LIN {X 80.299,Y 11.763,Z 59.815,A 180.000,B 0.000,C 180.000} C_DIS
LIN {X 80.187,Y 11.652,Z 59.809,A 180.000,B 0.000,C 180.000} C_DIS
LIN {X 80.132,Y 11.596,Z 59.806,A 180.000,B 0.000,C 180.000} C_DIS
LIN {X 80.020,Y 11.485,Z 59.801,A 180.000,B 0.000,C 180.000} C_DIS
LIN {X 79.853,Y 11.318,Z 59.793,A 180.000,B 0.000,C 180.000} C_DIS
LIN {X 79.742,Y 11.206,Z 59.787,A 180.000,B 0.000,C 180.000} C_DIS
LIN {X 79.686,Y 11.151,Z 59.785,A 180.000,B 0.000,C 180.000} C_DIS
LIN {X 79.575,Y 11.039,Z 59.779,A 180.000,B 0.000,C 180.000} C_DIS
LIN {X 79.408,Y 10.872,Z 59.771,A 180.000,B 0.000,C 180.000} C_DIS
LIN {X 79.296,Y 10.761,Z 59.765,A 180.000,B 0.000,C 180.000} C_DIS
LIN {X 79.241,Y 10.705,Z 59.763,A 180.000,B 0.000,C 180.000} C_DIS
LIN {X 79.183,Y 10.652,Z 59.760,A 180.000,B 0.000,C 180.000} C_DIS
LIN {X 79.124,Y 10.599,Z 59.757,A 180.000,B 0.000,C 180.000} C_DIS
LIN {X 79.063,Y 10.549,Z 59.754,A 180.000,B 0.000,C 180.000} C_DIS
LIN {X 79.001,Y 10.501,Z 59.752,A 180.000,B 0.000,C 180.000} C_DIS
LIN {X 78.938,Y 10.455,Z 59.749,A 180.000,B 0.000,C 180.000} C_DIS
LIN {X 78.872,Y 10.410,Z 59.746,A 180.000,B 0.000,C 180.000} C_DIS
LIN {X 78.806,Y 10.368,Z 59.743,A 180.000,B 0.000,C 180.000} C_DIS
LIN {X 78.738,Y 10.328,Z 59.741,A 180.000,B 0.000,C 180.000} C_DIS
LIN {X 78.669,Y 10.290,Z 59.738,A 180.000,B 0.000,C 180.000} C_DIS
LIN {X 78.599,Y 10.254,Z 59.735,A 180.000,B 0.000,C 180.000} C_DIS
LIN {X 78.528,Y 10.221,Z 59.732,A 180.000,B 0.000,C 180.000} C_DIS
LIN {X 78.455,Y 10.190,Z 59.730,A 180.000,B 0.000,C 180.000} C_DIS
LIN {X 78.382,Y 10.161,Z 59.727,A 180.000,B 0.000,C 180.000} C_DIS
LIN {X 78.308,Y 10.134,Z 59.724,A 180.000,B 0.000,C 180.000} C_DIS
LIN {X 78.233,Y 10.110,Z 59.721,A 180.000,B 0.000,C 180.000} C_DIS
LIN {X 78.157,Y 10.088,Z 59.719,A 180.000,B 0.000,C 180.000} C_DIS
LIN {X 78.081,Y 10.068,Z 59.716,A 180.000,B 0.000,C 180.000} C_DIS
LIN {X 78.004,Y 10.051,Z 59.713,A 180.000,B 0.000,C 180.000} C_DIS
LIN {X 77.927,Y 10.037,Z 59.710,A 180.000,B 0.000,C 180.000} C_DIS
LIN {X 77.849,Y 10.024,Z 59.708,A 180.000,B 0.000,C 180.000} C_DIS
LIN {X 77.771,Y 10.015,Z 59.705,A 180.000,B 0.000,C 180.000} C_DIS
LIN {X 77.692,Y 10.007,Z 59.702,A 180.000,B 0.000,C 180.000} C_DIS
LIN {X 77.614,Y 10.003,Z 59.699,A 180.000,B 0.000,C 180.000} C_DIS
LIN {X 77.535,Y 10.000,Z 59.697,A 180.000,B 0.000,C 180.000} C_DIS
LIN {X 77.456,Y 10.000,Z 59.694,A 180.000,B 0.000,C 180.000} C_DIS
LIN {X 77.377,Y 10.003,Z 59.691,A 180.000,B 0.000,C 180.000} C_DIS
LIN {X 77.299,Y 10.008,Z 59.688,A 180.000,B 0.000,C 180.000} C_DIS
LIN {X 77.220,Y 10.016,Z 59.686,A 180.000,B 0.000,C 180.000} C_DIS
LIN {X 77.142,Y 10.026,Z 59.683,A 180.000,B 0.000,C 180.000} C_DIS
LIN {X 77.065,Y 10.038,Z 59.680,A 180.000,B 0.000,C 180.000} C_DIS
LIN {X 76.987,Y 10.053,Z 59.677,A 180.000,B 0.000,C 180.000} C_DIS
LIN {X 76.910,Y 10.071,Z 59.675,A 180.000,B 0.000,C 180.000} C_DIS
LIN {X 76.834,Y 10.090,Z 59.672,A 180.000,B 0.000,C 180.000} C_DIS
LIN {X 76.759,Y 10.112,Z 59.669,A 180.000,B 0.000,C 180.000} C_DIS
LIN {X 76.684,Y 10.137,Z 59.666,A 180.000,B 0.000,C 180.000} C_DIS
LIN {X 76.610,Y 10.164,Z 59.664,A 180.000,B 0.000,C 180.000} C_DIS
LIN {X 76.537,Y 10.193,Z 59.661,A 180.000,B 0.000,C 180.000} C_DIS
LIN {X 76.464,Y 10.225,Z 59.658,A 180.000,B 0.000,C 180.000} C_DIS
LIN {X 76.393,Y 10.258,Z 59.655,A 180.000,B 0.000,C 180.000} C_DIS
LIN {X 76.323,Y 10.294,Z 59.653,A 180.000,B 0.000,C 180.000} C_DIS
LIN {X 76.254,Y 10.332,Z 59.650,A 180.000,B 0.000,C 180.000} C_DIS
LIN {X 76.187,Y 10.373,Z 59.647,A 180.000,B 0.000,C 180.000} C_DIS
LIN {X 76.120,Y 10.415,Z 59.644,A 180.000,B 0.000,C 180.000} C_DIS
LIN {X 76.055,Y 10.460,Z 59.642,A 180.000,B 0.000,C 180.000} C_DIS
LIN {X 75.992,Y 10.506,Z 59.639,A 180.000,B 0.000,C 180.000} C_DIS
LIN {X 75.930,Y 10.555,Z 59.636,A 180.000,B 0.000,C 180.000} C_DIS
LIN {X 75.869,Y 10.605,Z 59.633,A 180.000,B 0.000,C 180.000} C_DIS
LIN {X 75.810,Y 10.658,Z 59.631,A 180.000,B 0.000,C 180.000} C_DIS
LIN {X 75.753,Y 10.712,Z 59.628,A 180.000,B 0.000,C 180.000} C_DIS
LIN {X 75.697,Y 10.767,Z 59.625,A 180.000,B 0.000,C 180.000} C_DIS
LIN {X 75.140,Y 11.324,Z 59.598,A 180.000,B 0.000,C 180.000} C_DIS
LIN {X 74.973,Y 11.491,Z 59.589,A 180.000,B 0.000,C 180.000} C_DIS
LIN {X 74.751,Y 11.714,Z 59.578,A 180.000,B 0.000,C 180.000} C_DIS
LIN {X 74.472,Y 11.992,Z 59.565,A 180.000,B 0.000,C 180.000} C_DIS
LIN {X 74.138,Y 12.326,Z 59.548,A 180.000,B 0.000,C 180.000} C_DIS
LIN {X 72.857,Y 13.607,Z 59.485,A 180.000,B 0.000,C 180.000} C_DIS
LIN {X 70.741,Y 15.723,Z 59.380,A 180.000,B 0.000,C 180.000} C_DIS
LIN {X 70.630,Y 15.834,Z 59.375,A 180.000,B 0.000,C 180.000} C_DIS
LIN {X 70.296,Y 16.169,Z 59.358,A 180.000,B 0.000,C 180.000} C_DIS
LIN {X 70.185,Y 16.280,Z 59.353,A 180.000,B 0.000,C 180.000} C_DIS
LIN {X 69.850,Y 16.614,Z 59.336,A 180.000,B 0.000,C 180.000} C_DIS
LIN {X 69.795,Y 16.670,Z 59.334,A 180.000,B 0.000,C 180.000} C_DIS
LIN {X 69.683,Y 16.781,Z 59.328,A 180.000,B 0.000,C 180.000} C_DIS
LIN {X 69.349,Y 17.115,Z 59.312,A 180.000,B 0.000,C 180.000} C_DIS
LIN {X 69.238,Y 17.227,Z 59.306,A 180.000,B 0.000,C 180.000} C_DIS
LIN {X 68.904,Y 17.561,Z 59.290,A 180.000,B 0.000,C 180.000} C_DIS
LIN {X 68.792,Y 17.672,Z 59.284,A 180.000,B 0.000,C 180.000} C_DIS
LIN {X 68.625,Y 17.839,Z 59.276,A 180.000,B 0.000,C 180.000} C_DIS
LIN {X 68.514,Y 17.951,Z 59.270,A 180.000,B 0.000,C 180.000} C_DIS
LIN {X 68.458,Y 18.006,Z 59.268,A 180.000,B 0.000,C 180.000} C_DIS
LIN {X 68.347,Y 18.118,Z 59.262,A 180.000,B 0.000,C 180.000} C_DIS
LIN {X 68.180,Y 18.285,Z 59.254,A 180.000,B 0.000,C 180.000} C_DIS
LIN {X 68.068,Y 18.396,Z 59.248,A 180.000,B 0.000,C 180.000} C_DIS
LIN {X 68.013,Y 18.452,Z 59.246,A 180.000,B 0.000,C 180.000} C_DIS
LIN {X 67.901,Y 18.563,Z 59.240,A 180.000,B 0.000,C 180.000} C_DIS
LIN {X 67.734,Y 18.730,Z 59.232,A 180.000,B 0.000,C 180.000} C_DIS
LIN {X 67.623,Y 18.841,Z 59.226,A 180.000,B 0.000,C 180.000} C_DIS
LIN {X 67.567,Y 18.897,Z 59.224,A 180.000,B 0.000,C 180.000} C_DIS
LIN {X 67.456,Y 19.009,Z 59.218,A 180.000,B 0.000,C 180.000} C_DIS
LIN {X 67.289,Y 19.176,Z 59.210,A 180.000,B 0.000,C 180.000} C_DIS
LIN {X 67.178,Y 19.287,Z 59.204,A 180.000,B 0.000,C 180.000} C_DIS
LIN {X 67.122,Y 19.343,Z 59.202,A 180.000,B 0.000,C 180.000} C_DIS
LIN {X 67.010,Y 19.454,Z 59.196,A 180.000,B 0.000,C 180.000} C_DIS
LIN {X 66.899,Y 19.565,Z 59.191,A 180.000,B 0.000,C 180.000} C_DIS
LIN {X 66.788,Y 19.677,Z 59.185,A 180.000,B 0.000,C 180.000} C_DIS
LIN {X 66.676,Y 19.788,Z 59.180,A 180.000,B 0.000,C 180.000} C_DIS
LIN {X 66.565,Y 19.899,Z 59.174,A 180.000,B 0.000,C 180.000} C_DIS
LIN {X 66.454,Y 20.011,Z 59.169,A 180.000,B 0.000,C 180.000} C_DIS
LIN {X 66.342,Y 20.122,Z 59.164,A 180.000,B 0.000,C 180.000} C_DIS
LIN {X 66.287,Y 20.178,Z 59.161,A 180.000,B 0.000,C 180.000} C_DIS
LIN {X 66.231,Y 20.234,Z 59.159,A 180.000,B 0.000,C 180.000} C_DIS
LIN {X 66.175,Y 20.289,Z 59.156,A 180.000,B 0.000,C 180.000} C_DIS
LIN {X 66.120,Y 20.345,Z 59.154,A 180.000,B 0.000,C 180.000} C_DIS
LIN {X 66.064,Y 20.401,Z 59.151,A 180.000,B 0.000,C 180.000} C_DIS
LIN {X 66.008,Y 20.456,Z 59.149,A 180.000,B 0.000,C 180.000} C_DIS
LIN {X 65.897,Y 20.568,Z 59.144,A 180.000,B 0.000,C 180.000} C_DIS
LIN {X 65.785,Y 20.679,Z 59.139,A 180.000,B 0.000,C 180.000} C_DIS
LIN {X 65.674,Y 20.790,Z 59.134,A 180.000,B 0.000,C 180.000} C_DIS
LIN {X 65.563,Y 20.902,Z 59.129,A 180.000,B 0.000,C 180.000} C_DIS
LIN {X 65.451,Y 21.013,Z 59.124,A 180.000,B 0.000,C 180.000} C_DIS
LIN {X 65.340,Y 21.125,Z 59.120,A 180.000,B 0.000,C 180.000} C_DIS
LIN {X 65.229,Y 21.236,Z 59.115,A 180.000,B 0.000,C 180.000} C_DIS
LIN {X 65.117,Y 21.347,Z 59.111,A 180.000,B 0.000,C 180.000} C_DIS
LIN {X 65.006,Y 21.459,Z 59.106,A 180.000,B 0.000,C 180.000} C_DIS
LIN {X 64.894,Y 21.570,Z 59.102,A 180.000,B 0.000,C 180.000} C_DIS
LIN {X 64.783,Y 21.681,Z 59.097,A 180.000,B 0.000,C 180.000} C_DIS
LIN {X 64.672,Y 21.793,Z 59.093,A 180.000,B 0.000,C 180.000} C_DIS
LIN {X 64.560,Y 21.904,Z 59.089,A 180.000,B 0.000,C 180.000} C_DIS
LIN {X 64.449,Y 22.015,Z 59.085,A 180.000,B 0.000,C 180.000} C_DIS
LIN {X 64.338,Y 22.127,Z 59.081,A 180.000,B 0.000,C 180.000} C_DIS
LIN {X 64.226,Y 22.238,Z 59.077,A 180.000,B 0.000,C 180.000} C_DIS
LIN {X 64.115,Y 22.350,Z 59.073,A 180.000,B 0.000,C 180.000} C_DIS
LIN {X 64.004,Y 22.461,Z 59.070,A 180.000,B 0.000,C 180.000} C_DIS
LIN {X 63.892,Y 22.572,Z 59.066,A 180.000,B 0.000,C 180.000} C_DIS
LIN {X 63.781,Y 22.684,Z 59.062,A 180.000,B 0.000,C 180.000} C_DIS
LIN {X 63.669,Y 22.795,Z 59.059,A 180.000,B 0.000,C 180.000} C_DIS
LIN {X 63.558,Y 22.906,Z 59.056,A 180.000,B 0.000,C 180.000} C_DIS
LIN {X 63.447,Y 23.018,Z 59.052,A 180.000,B 0.000,C 180.000} C_DIS
LIN {X 63.335,Y 23.129,Z 59.049,A 180.000,B 0.000,C 180.000} C_DIS
LIN {X 63.224,Y 23.241,Z 59.046,A 180.000,B 0.000,C 180.000} C_DIS
LIN {X 63.113,Y 23.352,Z 59.043,A 180.000,B 0.000,C 180.000} C_DIS
LIN {X 63.001,Y 23.463,Z 59.040,A 180.000,B 0.000,C 180.000} C_DIS
LIN {X 62.890,Y 23.575,Z 59.037,A 180.000,B 0.000,C 180.000} C_DIS
LIN {X 62.778,Y 23.686,Z 59.034,A 180.000,B 0.000,C 180.000} C_DIS
LIN {X 62.667,Y 23.797,Z 59.032,A 180.000,B 0.000,C 180.000} C_DIS
LIN {X 62.556,Y 23.909,Z 59.029,A 180.000,B 0.000,C 180.000} C_DIS
LIN {X 62.444,Y 24.020,Z 59.027,A 180.000,B 0.000,C 180.000} C_DIS
LIN {X 62.222,Y 24.243,Z 59.022,A 180.000,B 0.000,C 180.000} C_DIS
LIN {X 61.999,Y 24.466,Z 59.018,A 180.000,B 0.000,C 180.000} C_DIS
LIN {X 61.776,Y 24.688,Z 59.014,A 180.000,B 0.000,C 180.000} C_DIS
LIN {X 61.553,Y 24.911,Z 59.011,A 180.000,B 0.000,C 180.000} C_DIS
LIN {X 61.331,Y 25.134,Z 59.008,A 180.000,B 0.000,C 180.000} C_DIS
LIN {X 61.108,Y 25.357,Z 59.005,A 180.000,B 0.000,C 180.000} C_DIS
LIN {X 60.885,Y 25.579,Z 59.003,A 180.000,B 0.000,C 180.000} C_DIS
LIN {X 60.662,Y 25.802,Z 59.002,A 180.000,B 0.000,C 180.000} C_DIS
LIN {X 60.440,Y 26.025,Z 59.001,A 180.000,B 0.000,C 180.000} C_DIS
LIN {X 60.217,Y 26.247,Z 59.000,A 180.000,B 0.000,C 180.000} C_DIS
LIN {X 60.053,Y 26.412,Z 59.000,A 180.000,B 0.000,C 180.000} C_DIS
; Cutting Move Starts
LIN {X 10.729,Y 75.735,Z 59.000,A 180.000,B 0.000,C 180.000} C_DIS
LIN {X 10.665,Y 75.802,Z 59.000,A 180.000,B 0.000,C 180.000} C_DIS
LIN {X 10.551,Y 75.935,Z 59.000,A 180.000,B 0.000,C 180.000} C_DIS
LIN {X 10.515,Y 75.980,Z 59.000,A 180.000,B 0.000,C 180.000} C_DIS
LIN {X 10.390,Y 76.159,Z 59.000,A 180.000,B 0.000,C 180.000} C_DIS
LIN {X 10.372,Y 76.188,Z 59.000,A 180.000,B 0.000,C 180.000} C_DIS
LIN {X 10.286,Y 76.338,Z 59.000,A 180.000,B 0.000,C 180.000} C_DIS
LIN {X 10.201,Y 76.517,Z 59.000,A 180.000,B 0.000,C 180.000} C_DIS
LIN {X 10.193,Y 76.537,Z 59.000,A 180.000,B 0.000,C 180.000} C_DIS
LIN {X 10.133,Y 76.696,Z 59.000,A 180.000,B 0.000,C 180.000} C_DIS
LIN {X 10.080,Y 76.874,Z 59.000,A 180.000,B 0.000,C 180.000} C_DIS
LIN {X 10.040,Y 77.053,Z 59.000,A 180.000,B 0.000,C 180.000} C_DIS
LIN {X 10.014,Y 77.232,Z 59.000,A 180.000,B 0.000,C 180.000} C_DIS
LIN {X 10.014,Y 77.233,Z 59.000,A 180.000,B 0.000,C 180.000} C_DIS
LIN {X 10.002,Y 77.411,Z 59.000,A 180.000,B 0.000,C 180.000} C_DIS
LIN {X 10.002,Y 77.589,Z 59.000,A 180.000,B 0.000,C 180.000} C_DIS
LIN {X 10.014,Y 77.767,Z 59.000,A 180.000,B 0.000,C 180.000} C_DIS
LIN {X 10.014,Y 77.768,Z 59.000,A 180.000,B 0.000,C 180.000} C_DIS
LIN {X 10.040,Y 77.947,Z 59.000,A 180.000,B 0.000,C 180.000} C_DIS
LIN {X 10.080,Y 78.126,Z 59.000,A 180.000,B 0.000,C 180.000} C_DIS
LIN {X 10.133,Y 78.304,Z 59.000,A 180.000,B 0.000,C 180.000} C_DIS
LIN {X 10.193,Y 78.463,Z 59.000,A 180.000,B 0.000,C 180.000} C_DIS
LIN {X 10.201,Y 78.483,Z 59.000,A 180.000,B 0.000,C 180.000} C_DIS
LIN {X 10.286,Y 78.662,Z 59.000,A 180.000,B 0.000,C 180.000} C_DIS
LIN {X 10.372,Y 78.812,Z 59.000,A 180.000,B 0.000,C 180.000} C_DIS
LIN {X 10.390,Y 78.841,Z 59.000,A 180.000,B 0.000,C 180.000} C_DIS
LIN {X 10.515,Y 79.020,Z 59.000,A 180.000,B 0.000,C 180.000} C_DIS
LIN {X 10.551,Y 79.065,Z 59.000,A 180.000,B 0.000,C 180.000} C_DIS
LIN {X 10.665,Y 79.198,Z 59.000,A 180.000,B 0.000,C 180.000} C_DIS
LIN {X 10.729,Y 79.265,Z 59.000,A 180.000,B 0.000,C 180.000} C_DIS
LIN {X 75.735,Y 144.271,Z 59.000,A 180.000,B 0.000,C 180.000} C_DIS
LIN {X 75.802,Y 144.335,Z 59.000,A 180.000,B 0.000,C 180.000} C_DIS
LIN {X 75.935,Y 144.449,Z 59.000,A 180.000,B 0.000,C 180.000} C_DIS
LIN {X 75.980,Y 144.485,Z 59.000,A 180.000,B 0.000,C 180.000} C_DIS
LIN {X 76.159,Y 144.610,Z 59.000,A 180.000,B 0.000,C 180.000} C_DIS
LIN {X 76.188,Y 144.628,Z 59.000,A 180.000,B 0.000,C 180.000} C_DIS
LIN {X 76.338,Y 144.714,Z 59.000,A 180.000,B 0.000,C 180.000} C_DIS
LIN {X 76.517,Y 144.799,Z 59.000,A 180.000,B 0.000,C 180.000} C_DIS
LIN {X 76.537,Y 144.807,Z 59.000,A 180.000,B 0.000,C 180.000} C_DIS
LIN {X 76.696,Y 144.867,Z 59.000,A 180.000,B 0.000,C 180.000} C_DIS
LIN {X 76.874,Y 144.920,Z 59.000,A 180.000,B 0.000,C 180.000} C_DIS
LIN {X 77.053,Y 144.960,Z 59.000,A 180.000,B 0.000,C 180.000} C_DIS
LIN {X 77.232,Y 144.986,Z 59.000,A 180.000,B 0.000,C 180.000} C_DIS
LIN {X 77.233,Y 144.986,Z 59.000,A 180.000,B 0.000,C 180.000} C_DIS
LIN {X 77.411,Y 144.998,Z 59.000,A 180.000,B 0.000,C 180.000} C_DIS
LIN {X 77.589,Y 144.998,Z 59.000,A 180.000,B 0.000,C 180.000} C_DIS
LIN {X 77.767,Y 144.986,Z 59.000,A 180.000,B 0.000,C 180.000} C_DIS
LIN {X 77.768,Y 144.986,Z 59.000,A 180.000,B 0.000,C 180.000} C_DIS
LIN {X 77.947,Y 144.960,Z 59.000,A 180.000,B 0.000,C 180.000} C_DIS
LIN {X 78.126,Y 144.920,Z 59.000,A 180.000,B 0.000,C 180.000} C_DIS
LIN {X 78.304,Y 144.867,Z 59.000,A 180.000,B 0.000,C 180.000} C_DIS
LIN {X 78.463,Y 144.807,Z 59.000,A 180.000,B 0.000,C 180.000} C_DIS
LIN {X 78.483,Y 144.799,Z 59.000,A 180.000,B 0.000,C 180.000} C_DIS
LIN {X 78.662,Y 144.714,Z 59.000,A 180.000,B 0.000,C 180.000} C_DIS
LIN {X 78.812,Y 144.628,Z 59.000,A 180.000,B 0.000,C 180.000} C_DIS
LIN {X 78.841,Y 144.610,Z 59.000,A 180.000,B 0.000,C 180.000} C_DIS
LIN {X 79.020,Y 144.485,Z 59.000,A 180.000,B 0.000,C 180.000} C_DIS
LIN {X 79.065,Y 144.449,Z 59.000,A 180.000,B 0.000,C 180.000} C_DIS
LIN {X 79.198,Y 144.335,Z 59.000,A 180.000,B 0.000,C 180.000} C_DIS
LIN {X 79.265,Y 144.271,Z 59.000,A 180.000,B 0.000,C 180.000} C_DIS
LIN {X 144.271,Y 79.265,Z 59.000,A 180.000,B 0.000,C 180.000} C_DIS
LIN {X 144.335,Y 79.198,Z 59.000,A 180.000,B 0.000,C 180.000} C_DIS
LIN {X 144.449,Y 79.065,Z 59.000,A 180.000,B 0.000,C 180.000} C_DIS
LIN {X 144.485,Y 79.020,Z 59.000,A 180.000,B 0.000,C 180.000} C_DIS
LIN {X 144.610,Y 78.841,Z 59.000,A 180.000,B 0.000,C 180.000} C_DIS
LIN {X 144.628,Y 78.812,Z 59.000,A 180.000,B 0.000,C 180.000} C_DIS
LIN {X 144.714,Y 78.662,Z 59.000,A 180.000,B 0.000,C 180.000} C_DIS
LIN {X 144.799,Y 78.483,Z 59.000,A 180.000,B 0.000,C 180.000} C_DIS
LIN {X 144.807,Y 78.463,Z 59.000,A 180.000,B 0.000,C 180.000} C_DIS
LIN {X 144.867,Y 78.304,Z 59.000,A 180.000,B 0.000,C 180.000} C_DIS
LIN {X 144.920,Y 78.126,Z 59.000,A 180.000,B 0.000,C 180.000} C_DIS
LIN {X 144.960,Y 77.947,Z 59.000,A 180.000,B 0.000,C 180.000} C_DIS
LIN {X 144.986,Y 77.768,Z 59.000,A 180.000,B 0.000,C 180.000} C_DIS
LIN {X 144.986,Y 77.767,Z 59.000,A 180.000,B 0.000,C 180.000} C_DIS
LIN {X 144.998,Y 77.589,Z 59.000,A 180.000,B 0.000,C 180.000} C_DIS
LIN {X 144.998,Y 77.411,Z 59.000,A 180.000,B 0.000,C 180.000} C_DIS
LIN {X 144.986,Y 77.233,Z 59.000,A 180.000,B 0.000,C 180.000} C_DIS
LIN {X 144.986,Y 77.232,Z 59.000,A 180.000,B 0.000,C 180.000} C_DIS
LIN {X 144.960,Y 77.053,Z 59.000,A 180.000,B 0.000,C 180.000} C_DIS
LIN {X 144.920,Y 76.874,Z 59.000,A 180.000,B 0.000,C 180.000} C_DIS
LIN {X 144.867,Y 76.696,Z 59.000,A 180.000,B 0.000,C 180.000} C_DIS
LIN {X 144.807,Y 76.537,Z 59.000,A 180.000,B 0.000,C 180.000} C_DIS
LIN {X 144.799,Y 76.517,Z 59.000,A 180.000,B 0.000,C 180.000} C_DIS
LIN {X 144.714,Y 76.338,Z 59.000,A 180.000,B 0.000,C 180.000} C_DIS
LIN {X 144.628,Y 76.188,Z 59.000,A 180.000,B 0.000,C 180.000} C_DIS
LIN {X 144.610,Y 76.159,Z 59.000,A 180.000,B 0.000,C 180.000} C_DIS
LIN {X 144.485,Y 75.980,Z 59.000,A 180.000,B 0.000,C 180.000} C_DIS
LIN {X 144.449,Y 75.935,Z 59.000,A 180.000,B 0.000,C 180.000} C_DIS
LIN {X 144.335,Y 75.802,Z 59.000,A 180.000,B 0.000,C 180.000} C_DIS
LIN {X 144.271,Y 75.735,Z 59.000,A 180.000,B 0.000,C 180.000} C_DIS
LIN {X 109.686,Y 41.150,Z 59.000,A 180.000,B 0.000,C 180.000} C_DIS
LIN {X 87.037,Y 18.501,Z 59.000,A 180.000,B 0.000,C 180.000} C_DIS
LIN {X 79.265,Y 10.729,Z 59.000,A 180.000,B 0.000,C 180.000} C_DIS
LIN {X 79.198,Y 10.665,Z 59.000,A 180.000,B 0.000,C 180.000} C_DIS
LIN {X 79.065,Y 10.551,Z 59.000,A 180.000,B 0.000,C 180.000} C_DIS
LIN {X 79.020,Y 10.515,Z 59.000,A 180.000,B 0.000,C 180.000} C_DIS
LIN {X 78.841,Y 10.390,Z 59.000,A 180.000,B 0.000,C 180.000} C_DIS
LIN {X 78.812,Y 10.372,Z 59.000,A 180.000,B 0.000,C 180.000} C_DIS
LIN {X 78.662,Y 10.286,Z 59.000,A 180.000,B 0.000,C 180.000} C_DIS
LIN {X 78.483,Y 10.201,Z 59.000,A 180.000,B 0.000,C 180.000} C_DIS
LIN {X 78.463,Y 10.193,Z 59.000,A 180.000,B 0.000,C 180.000} C_DIS
LIN {X 78.304,Y 10.133,Z 59.000,A 180.000,B 0.000,C 180.000} C_DIS
LIN {X 78.126,Y 10.080,Z 59.000,A 180.000,B 0.000,C 180.000} C_DIS
LIN {X 77.947,Y 10.040,Z 59.000,A 180.000,B 0.000,C 180.000} C_DIS
LIN {X 77.768,Y 10.014,Z 59.000,A 180.000,B 0.000,C 180.000} C_DIS
LIN {X 77.767,Y 10.014,Z 59.000,A 180.000,B 0.000,C 180.000} C_DIS
LIN {X 77.589,Y 10.002,Z 59.000,A 180.000,B 0.000,C 180.000} C_DIS
LIN {X 77.411,Y 10.002,Z 59.000,A 180.000,B 0.000,C 180.000} C_DIS
LIN {X 77.233,Y 10.014,Z 59.000,A 180.000,B 0.000,C 180.000} C_DIS
LIN {X 77.232,Y 10.014,Z 59.000,A 180.000,B 0.000,C 180.000} C_DIS
LIN {X 77.053,Y 10.040,Z 59.000,A 180.000,B 0.000,C 180.000} C_DIS
LIN {X 76.874,Y 10.080,Z 59.000,A 180.000,B 0.000,C 180.000} C_DIS
LIN {X 76.696,Y 10.133,Z 59.000,A 180.000,B 0.000,C 180.000} C_DIS
LIN {X 76.537,Y 10.193,Z 59.000,A 180.000,B 0.000,C 180.000} C_DIS
LIN {X 76.517,Y 10.201,Z 59.000,A 180.000,B 0.000,C 180.000} C_DIS
LIN {X 76.338,Y 10.286,Z 59.000,A 180.000,B 0.000,C 180.000} C_DIS
LIN {X 76.188,Y 10.372,Z 59.000,A 180.000,B 0.000,C 180.000} C_DIS
LIN {X 76.159,Y 10.390,Z 59.000,A 180.000,B 0.000,C 180.000} C_DIS
LIN {X 75.980,Y 10.515,Z 59.000,A 180.000,B 0.000,C 180.000} C_DIS
LIN {X 75.935,Y 10.551,Z 59.000,A 180.000,B 0.000,C 180.000} C_DIS
LIN {X 75.802,Y 10.665,Z 59.000,A 180.000,B 0.000,C 180.000} C_DIS
LIN {X 75.735,Y 10.729,Z 59.000,A 180.000,B 0.000,C 180.000} C_DIS
LIN {X 60.053,Y 26.412,Z 59.000,A 180.000,B 0.000,C 180.000} C_DIS
; Link Move Starts
LIN {X 59.830,Y 26.635,Z 59.000,A 180.000,B 0.000,C 180.000} C_DIS
LIN {X 59.607,Y 26.857,Z 58.999,A 180.000,B 0.000,C 180.000} C_DIS
LIN {X 59.384,Y 27.080,Z 58.998,A 180.000,B 0.000,C 180.000} C_DIS
LIN {X 59.162,Y 27.303,Z 58.996,A 180.000,B 0.000,C 180.000} C_DIS
LIN {X 58.939,Y 27.526,Z 58.994,A 180.000,B 0.000,C 180.000} C_DIS
LIN {X 58.716,Y 27.748,Z 58.991,A 180.000,B 0.000,C 180.000} C_DIS
LIN {X 58.493,Y 27.971,Z 58.988,A 180.000,B 0.000,C 180.000} C_DIS
LIN {X 58.271,Y 28.194,Z 58.985,A 180.000,B 0.000,C 180.000} C_DIS
LIN {X 58.048,Y 28.417,Z 58.981,A 180.000,B 0.000,C 180.000} C_DIS
LIN {X 57.825,Y 28.639,Z 58.977,A 180.000,B 0.000,C 180.000} C_DIS
LIN {X 57.602,Y 28.862,Z 58.972,A 180.000,B 0.000,C 180.000} C_DIS
LIN {X 57.491,Y 28.973,Z 58.969,A 180.000,B 0.000,C 180.000} C_DIS
LIN {X 57.380,Y 29.085,Z 58.967,A 180.000,B 0.000,C 180.000} C_DIS
LIN {X 57.268,Y 29.196,Z 58.964,A 180.000,B 0.000,C 180.000} C_DIS
LIN {X 57.157,Y 29.308,Z 58.961,A 180.000,B 0.000,C 180.000} C_DIS
LIN {X 57.046,Y 29.419,Z 58.959,A 180.000,B 0.000,C 180.000} C_DIS
LIN {X 56.934,Y 29.530,Z 58.956,A 180.000,B 0.000,C 180.000} C_DIS
LIN {X 56.823,Y 29.642,Z 58.952,A 180.000,B 0.000,C 180.000} C_DIS
LIN {X 56.711,Y 29.753,Z 58.949,A 180.000,B 0.000,C 180.000} C_DIS
LIN {X 56.600,Y 29.864,Z 58.946,A 180.000,B 0.000,C 180.000} C_DIS
LIN {X 56.489,Y 29.976,Z 58.943,A 180.000,B 0.000,C 180.000} C_DIS
LIN {X 56.377,Y 30.087,Z 58.939,A 180.000,B 0.000,C 180.000} C_DIS
LIN {X 56.266,Y 30.198,Z 58.936,A 180.000,B 0.000,C 180.000} C_DIS
LIN {X 56.155,Y 30.310,Z 58.932,A 180.000,B 0.000,C 180.000} C_DIS
LIN {X 56.043,Y 30.421,Z 58.928,A 180.000,B 0.000,C 180.000} C_DIS
LIN {X 55.932,Y 30.533,Z 58.925,A 180.000,B 0.000,C 180.000} C_DIS
LIN {X 55.820,Y 30.644,Z 58.921,A 180.000,B 0.000,C 180.000} C_DIS
LIN {X 55.709,Y 30.755,Z 58.917,A 180.000,B 0.000,C 180.000} C_DIS
LIN {X 55.598,Y 30.867,Z 58.913,A 180.000,B 0.000,C 180.000} C_DIS
LIN {X 55.486,Y 30.978,Z 58.909,A 180.000,B 0.000,C 180.000} C_DIS
LIN {X 55.375,Y 31.089,Z 58.905,A 180.000,B 0.000,C 180.000} C_DIS
LIN {X 55.264,Y 31.201,Z 58.900,A 180.000,B 0.000,C 180.000} C_DIS
LIN {X 55.152,Y 31.312,Z 58.896,A 180.000,B 0.000,C 180.000} C_DIS
LIN {X 55.041,Y 31.424,Z 58.892,A 180.000,B 0.000,C 180.000} C_DIS
LIN {X 54.930,Y 31.535,Z 58.887,A 180.000,B 0.000,C 180.000} C_DIS
LIN {X 54.818,Y 31.646,Z 58.883,A 180.000,B 0.000,C 180.000} C_DIS
LIN {X 54.707,Y 31.758,Z 58.878,A 180.000,B 0.000,C 180.000} C_DIS
LIN {X 54.595,Y 31.869,Z 58.873,A 180.000,B 0.000,C 180.000} C_DIS
LIN {X 54.484,Y 31.980,Z 58.869,A 180.000,B 0.000,C 180.000} C_DIS
LIN {X 54.373,Y 32.092,Z 58.864,A 180.000,B 0.000,C 180.000} C_DIS
LIN {X 54.261,Y 32.203,Z 58.859,A 180.000,B 0.000,C 180.000} C_DIS
LIN {X 54.150,Y 32.315,Z 58.854,A 180.000,B 0.000,C 180.000} C_DIS
LIN {X 54.094,Y 32.370,Z 58.851,A 180.000,B 0.000,C 180.000} C_DIS
LIN {X 54.039,Y 32.426,Z 58.849,A 180.000,B 0.000,C 180.000} C_DIS
LIN {X 53.983,Y 32.482,Z 58.846,A 180.000,B 0.000,C 180.000} C_DIS
LIN {X 53.927,Y 32.537,Z 58.844,A 180.000,B 0.000,C 180.000} C_DIS
LIN {X 53.872,Y 32.593,Z 58.841,A 180.000,B 0.000,C 180.000} C_DIS
LIN {X 53.816,Y 32.649,Z 58.839,A 180.000,B 0.000,C 180.000} C_DIS
LIN {X 53.760,Y 32.704,Z 58.836,A 180.000,B 0.000,C 180.000} C_DIS
LIN {X 53.649,Y 32.816,Z 58.831,A 180.000,B 0.000,C 180.000} C_DIS
LIN {X 53.537,Y 32.927,Z 58.825,A 180.000,B 0.000,C 180.000} C_DIS
LIN {X 53.426,Y 33.038,Z 58.820,A 180.000,B 0.000,C 180.000} C_DIS
LIN {X 53.315,Y 33.150,Z 58.815,A 180.000,B 0.000,C 180.000} C_DIS
LIN {X 53.203,Y 33.261,Z 58.809,A 180.000,B 0.000,C 180.000} C_DIS
LIN {X 53.148,Y 33.317,Z 58.806,A 180.000,B 0.000,C 180.000} C_DIS
LIN {X 53.036,Y 33.428,Z 58.801,A 180.000,B 0.000,C 180.000} C_DIS
LIN {X 52.869,Y 33.595,Z 58.793,A 180.000,B 0.000,C 180.000} C_DIS
LIN {X 52.758,Y 33.707,Z 58.787,A 180.000,B 0.000,C 180.000} C_DIS
LIN {X 52.702,Y 33.762,Z 58.785,A 180.000,B 0.000,C 180.000} C_DIS
LIN {X 52.591,Y 33.874,Z 58.779,A 180.000,B 0.000,C 180.000} C_DIS
LIN {X 52.424,Y 34.041,Z 58.771,A 180.000,B 0.000,C 180.000} C_DIS
LIN {X 52.312,Y 34.152,Z 58.765,A 180.000,B 0.000,C 180.000} C_DIS
LIN {X 52.257,Y 34.208,Z 58.763,A 180.000,B 0.000,C 180.000} C_DIS
LIN {X 52.145,Y 34.319,Z 58.757,A 180.000,B 0.000,C 180.000} C_DIS
LIN {X 51.978,Y 34.486,Z 58.749,A 180.000,B 0.000,C 180.000} C_DIS
LIN {X 51.867,Y 34.598,Z 58.743,A 180.000,B 0.000,C 180.000} C_DIS
LIN {X 51.811,Y 34.653,Z 58.741,A 180.000,B 0.000,C 180.000} C_DIS
LIN {X 51.700,Y 34.765,Z 58.735,A 180.000,B 0.000,C 180.000} C_DIS
LIN {X 51.533,Y 34.932,Z 58.727,A 180.000,B 0.000,C 180.000} C_DIS
LIN {X 51.421,Y 35.043,Z 58.721,A 180.000,B 0.000,C 180.000} C_DIS
LIN {X 51.366,Y 35.099,Z 58.719,A 180.000,B 0.000,C 180.000} C_DIS
LIN {X 51.254,Y 35.210,Z 58.713,A 180.000,B 0.000,C 180.000} C_DIS
LIN {X 50.920,Y 35.544,Z 58.697,A 180.000,B 0.000,C 180.000} C_DIS
LIN {X 50.809,Y 35.656,Z 58.691,A 180.000,B 0.000,C 180.000} C_DIS
LIN {X 50.475,Y 35.990,Z 58.675,A 180.000,B 0.000,C 180.000} C_DIS
LIN {X 50.363,Y 36.101,Z 58.669,A 180.000,B 0.000,C 180.000} C_DIS
LIN {X 49.974,Y 36.491,Z 58.650,A 180.000,B 0.000,C 180.000} C_DIS
LIN {X 49.640,Y 36.825,Z 58.633,A 180.000,B 0.000,C 180.000} C_DIS
LIN {X 49.528,Y 36.936,Z 58.628,A 180.000,B 0.000,C 180.000} C_DIS
LIN {X 49.194,Y 37.270,Z 58.611,A 180.000,B 0.000,C 180.000} C_DIS
LIN {X 49.083,Y 37.382,Z 58.606,A 180.000,B 0.000,C 180.000} C_DIS
LIN {X 48.526,Y 37.939,Z 58.578,A 180.000,B 0.000,C 180.000} C_DIS
LIN {X 48.247,Y 38.217,Z 58.565,A 180.000,B 0.000,C 180.000} C_DIS
LIN {X 47.913,Y 38.551,Z 58.548,A 180.000,B 0.000,C 180.000} C_DIS
LIN {X 46.633,Y 39.832,Z 58.485,A 180.000,B 0.000,C 180.000} C_DIS
LIN {X 44.517,Y 41.948,Z 58.380,A 180.000,B 0.000,C 180.000} C_DIS
LIN {X 44.405,Y 42.059,Z 58.375,A 180.000,B 0.000,C 180.000} C_DIS
LIN {X 44.071,Y 42.393,Z 58.358,A 180.000,B 0.000,C 180.000} C_DIS
LIN {X 43.960,Y 42.505,Z 58.353,A 180.000,B 0.000,C 180.000} C_DIS
LIN {X 43.626,Y 42.839,Z 58.336,A 180.000,B 0.000,C 180.000} C_DIS
LIN {X 43.570,Y 42.895,Z 58.334,A 180.000,B 0.000,C 180.000} C_DIS
LIN {X 43.459,Y 43.006,Z 58.328,A 180.000,B 0.000,C 180.000} C_DIS
LIN {X 43.124,Y 43.340,Z 58.312,A 180.000,B 0.000,C 180.000} C_DIS
LIN {X 43.013,Y 43.451,Z 58.306,A 180.000,B 0.000,C 180.000} C_DIS
LIN {X 42.679,Y 43.785,Z 58.290,A 180.000,B 0.000,C 180.000} C_DIS
LIN {X 42.568,Y 43.897,Z 58.284,A 180.000,B 0.000,C 180.000} C_DIS
LIN {X 42.401,Y 44.064,Z 58.276,A 180.000,B 0.000,C 180.000} C_DIS
LIN {X 42.289,Y 44.175,Z 58.270,A 180.000,B 0.000,C 180.000} C_DIS
LIN {X 42.233,Y 44.231,Z 58.268,A 180.000,B 0.000,C 180.000} C_DIS
LIN {X 42.122,Y 44.342,Z 58.262,A 180.000,B 0.000,C 180.000} C_DIS
LIN {X 41.955,Y 44.509,Z 58.254,A 180.000,B 0.000,C 180.000} C_DIS
LIN {X 41.844,Y 44.621,Z 58.248,A 180.000,B 0.000,C 180.000} C_DIS
LIN {X 41.788,Y 44.676,Z 58.246,A 180.000,B 0.000,C 180.000} C_DIS
LIN {X 41.677,Y 44.788,Z 58.240,A 180.000,B 0.000,C 180.000} C_DIS
LIN {X 41.510,Y 44.955,Z 58.232,A 180.000,B 0.000,C 180.000} C_DIS
LIN {X 41.398,Y 45.066,Z 58.226,A 180.000,B 0.000,C 180.000} C_DIS
LIN {X 41.343,Y 45.122,Z 58.224,A 180.000,B 0.000,C 180.000} C_DIS
LIN {X 41.231,Y 45.233,Z 58.218,A 180.000,B 0.000,C 180.000} C_DIS
LIN {X 41.064,Y 45.400,Z 58.210,A 180.000,B 0.000,C 180.000} C_DIS
LIN {X 40.953,Y 45.512,Z 58.204,A 180.000,B 0.000,C 180.000} C_DIS
LIN {X 40.897,Y 45.567,Z 58.202,A 180.000,B 0.000,C 180.000} C_DIS
LIN {X 40.786,Y 45.679,Z 58.196,A 180.000,B 0.000,C 180.000} C_DIS
LIN {X 40.674,Y 45.790,Z 58.191,A 180.000,B 0.000,C 180.000} C_DIS
LIN {X 40.563,Y 45.902,Z 58.185,A 180.000,B 0.000,C 180.000} C_DIS
LIN {X 40.452,Y 46.013,Z 58.180,A 180.000,B 0.000,C 180.000} C_DIS
LIN {X 40.340,Y 46.124,Z 58.174,A 180.000,B 0.000,C 180.000} C_DIS
LIN {X 40.229,Y 46.236,Z 58.169,A 180.000,B 0.000,C 180.000} C_DIS
LIN {X 40.117,Y 46.347,Z 58.164,A 180.000,B 0.000,C 180.000} C_DIS
LIN {X 40.062,Y 46.403,Z 58.161,A 180.000,B 0.000,C 180.000} C_DIS
LIN {X 40.006,Y 46.458,Z 58.159,A 180.000,B 0.000,C 180.000} C_DIS
LIN {X 39.950,Y 46.514,Z 58.156,A 180.000,B 0.000,C 180.000} C_DIS
LIN {X 39.895,Y 46.570,Z 58.154,A 180.000,B 0.000,C 180.000} C_DIS
LIN {X 39.839,Y 46.625,Z 58.151,A 180.000,B 0.000,C 180.000} C_DIS
LIN {X 39.783,Y 46.681,Z 58.148,A 180.000,B 0.000,C 180.000} C_DIS
LIN {X 39.672,Y 46.792,Z 58.143,A 180.000,B 0.000,C 180.000} C_DIS
LIN {X 39.561,Y 46.904,Z 58.139,A 180.000,B 0.000,C 180.000} C_DIS
LIN {X 39.449,Y 47.015,Z 58.134,A 180.000,B 0.000,C 180.000} C_DIS
LIN {X 39.338,Y 47.127,Z 58.129,A 180.000,B 0.000,C 180.000} C_DIS
LIN {X 39.227,Y 47.238,Z 58.124,A 180.000,B 0.000,C 180.000} C_DIS
LIN {X 39.115,Y 47.349,Z 58.120,A 180.000,B 0.000,C 180.000} C_DIS
LIN {X 39.004,Y 47.461,Z 58.115,A 180.000,B 0.000,C 180.000} C_DIS
LIN {X 38.892,Y 47.572,Z 58.110,A 180.000,B 0.000,C 180.000} C_DIS
LIN {X 38.781,Y 47.683,Z 58.106,A 180.000,B 0.000,C 180.000} C_DIS
LIN {X 38.670,Y 47.795,Z 58.102,A 180.000,B 0.000,C 180.000} C_DIS
LIN {X 38.558,Y 47.906,Z 58.097,A 180.000,B 0.000,C 180.000} C_DIS
LIN {X 38.447,Y 48.018,Z 58.093,A 180.000,B 0.000,C 180.000} C_DIS
LIN {X 38.336,Y 48.129,Z 58.089,A 180.000,B 0.000,C 180.000} C_DIS
LIN {X 38.224,Y 48.240,Z 58.085,A 180.000,B 0.000,C 180.000} C_DIS
LIN {X 38.113,Y 48.352,Z 58.081,A 180.000,B 0.000,C 180.000} C_DIS
LIN {X 38.001,Y 48.463,Z 58.077,A 180.000,B 0.000,C 180.000} C_DIS
LIN {X 37.890,Y 48.574,Z 58.073,A 180.000,B 0.000,C 180.000} C_DIS
LIN {X 37.779,Y 48.686,Z 58.070,A 180.000,B 0.000,C 180.000} C_DIS
LIN {X 37.667,Y 48.797,Z 58.066,A 180.000,B 0.000,C 180.000} C_DIS
LIN {X 37.556,Y 48.908,Z 58.062,A 180.000,B 0.000,C 180.000} C_DIS
LIN {X 37.445,Y 49.020,Z 58.059,A 180.000,B 0.000,C 180.000} C_DIS
LIN {X 37.333,Y 49.131,Z 58.056,A 180.000,B 0.000,C 180.000} C_DIS
LIN {X 37.222,Y 49.243,Z 58.052,A 180.000,B 0.000,C 180.000} C_DIS
LIN {X 37.111,Y 49.354,Z 58.049,A 180.000,B 0.000,C 180.000} C_DIS
LIN {X 36.999,Y 49.465,Z 58.046,A 180.000,B 0.000,C 180.000} C_DIS
LIN {X 36.888,Y 49.577,Z 58.043,A 180.000,B 0.000,C 180.000} C_DIS
LIN {X 36.776,Y 49.688,Z 58.040,A 180.000,B 0.000,C 180.000} C_DIS
LIN {X 36.665,Y 49.799,Z 58.037,A 180.000,B 0.000,C 180.000} C_DIS
LIN {X 36.554,Y 49.911,Z 58.034,A 180.000,B 0.000,C 180.000} C_DIS
LIN {X 36.442,Y 50.022,Z 58.032,A 180.000,B 0.000,C 180.000} C_DIS
LIN {X 36.331,Y 50.134,Z 58.029,A 180.000,B 0.000,C 180.000} C_DIS
LIN {X 36.220,Y 50.245,Z 58.027,A 180.000,B 0.000,C 180.000} C_DIS
LIN {X 35.997,Y 50.468,Z 58.022,A 180.000,B 0.000,C 180.000} C_DIS
LIN {X 35.774,Y 50.690,Z 58.018,A 180.000,B 0.000,C 180.000} C_DIS
LIN {X 35.551,Y 50.913,Z 58.014,A 180.000,B 0.000,C 180.000} C_DIS
LIN {X 35.329,Y 51.136,Z 58.011,A 180.000,B 0.000,C 180.000} C_DIS
LIN {X 35.106,Y 51.359,Z 58.008,A 180.000,B 0.000,C 180.000} C_DIS
LIN {X 34.883,Y 51.581,Z 58.005,A 180.000,B 0.000,C 180.000} C_DIS
LIN {X 34.660,Y 51.804,Z 58.003,A 180.000,B 0.000,C 180.000} C_DIS
LIN {X 34.438,Y 52.027,Z 58.002,A 180.000,B 0.000,C 180.000} C_DIS
LIN {X 34.215,Y 52.250,Z 58.001,A 180.000,B 0.000,C 180.000} C_DIS
LIN {X 33.992,Y 52.472,Z 58.000,A 180.000,B 0.000,C 180.000} C_DIS
LIN {X 33.829,Y 52.636,Z 58.000,A 180.000,B 0.000,C 180.000} C_DIS
; Cutting Move Starts
LIN {X 10.729,Y 75.735,Z 58.000,A 180.000,B 0.000,C 180.000} C_DIS
LIN {X 10.665,Y 75.802,Z 58.000,A 180.000,B 0.000,C 180.000} C_DIS
LIN {X 10.551,Y 75.935,Z 58.000,A 180.000,B 0.000,C 180.000} C_DIS
LIN {X 10.515,Y 75.980,Z 58.000,A 180.000,B 0.000,C 180.000} C_DIS
LIN {X 10.390,Y 76.159,Z 58.000,A 180.000,B 0.000,C 180.000} C_DIS
LIN {X 10.372,Y 76.188,Z 58.000,A 180.000,B 0.000,C 180.000} C_DIS
LIN {X 10.286,Y 76.338,Z 58.000,A 180.000,B 0.000,C 180.000} C_DIS
LIN {X 10.201,Y 76.517,Z 58.000,A 180.000,B 0.000,C 180.000} C_DIS
LIN {X 10.193,Y 76.537,Z 58.000,A 180.000,B 0.000,C 180.000} C_DIS
LIN {X 10.133,Y 76.696,Z 58.000,A 180.000,B 0.000,C 180.000} C_DIS
LIN {X 10.080,Y 76.874,Z 58.000,A 180.000,B 0.000,C 180.000} C_DIS
LIN {X 10.040,Y 77.053,Z 58.000,A 180.000,B 0.000,C 180.000} C_DIS
LIN {X 10.014,Y 77.232,Z 58.000,A 180.000,B 0.000,C 180.000} C_DIS
LIN {X 10.014,Y 77.233,Z 58.000,A 180.000,B 0.000,C 180.000} C_DIS
LIN {X 10.002,Y 77.411,Z 58.000,A 180.000,B 0.000,C 180.000} C_DIS
LIN {X 10.002,Y 77.589,Z 58.000,A 180.000,B 0.000,C 180.000} C_DIS
LIN {X 10.014,Y 77.767,Z 58.000,A 180.000,B 0.000,C 180.000} C_DIS
LIN {X 10.014,Y 77.768,Z 58.000,A 180.000,B 0.000,C 180.000} C_DIS
LIN {X 10.040,Y 77.947,Z 58.000,A 180.000,B 0.000,C 180.000} C_DIS
LIN {X 10.080,Y 78.126,Z 58.000,A 180.000,B 0.000,C 180.000} C_DIS
LIN {X 10.133,Y 78.304,Z 58.000,A 180.000,B 0.000,C 180.000} C_DIS
LIN {X 10.193,Y 78.463,Z 58.000,A 180.000,B 0.000,C 180.000} C_DIS
LIN {X 10.201,Y 78.483,Z 58.000,A 180.000,B 0.000,C 180.000} C_DIS
LIN {X 10.286,Y 78.662,Z 58.000,A 180.000,B 0.000,C 180.000} C_DIS
LIN {X 10.372,Y 78.812,Z 58.000,A 180.000,B 0.000,C 180.000} C_DIS
LIN {X 10.390,Y 78.841,Z 58.000,A 180.000,B 0.000,C 180.000} C_DIS
LIN {X 10.515,Y 79.020,Z 58.000,A 180.000,B 0.000,C 180.000} C_DIS
LIN {X 10.551,Y 79.065,Z 58.000,A 180.000,B 0.000,C 180.000} C_DIS
LIN {X 10.665,Y 79.198,Z 58.000,A 180.000,B 0.000,C 180.000} C_DIS
LIN {X 10.729,Y 79.265,Z 58.000,A 180.000,B 0.000,C 180.000} C_DIS
LIN {X 75.735,Y 144.271,Z 58.000,A 180.000,B 0.000,C 180.000} C_DIS
LIN {X 75.802,Y 144.335,Z 58.000,A 180.000,B 0.000,C 180.000} C_DIS
LIN {X 75.935,Y 144.449,Z 58.000,A 180.000,B 0.000,C 180.000} C_DIS
LIN {X 75.980,Y 144.485,Z 58.000,A 180.000,B 0.000,C 180.000} C_DIS
LIN {X 76.159,Y 144.610,Z 58.000,A 180.000,B 0.000,C 180.000} C_DIS
LIN {X 76.188,Y 144.628,Z 58.000,A 180.000,B 0.000,C 180.000} C_DIS
LIN {X 76.338,Y 144.714,Z 58.000,A 180.000,B 0.000,C 180.000} C_DIS
LIN {X 76.517,Y 144.799,Z 58.000,A 180.000,B 0.000,C 180.000} C_DIS
LIN {X 76.537,Y 144.807,Z 58.000,A 180.000,B 0.000,C 180.000} C_DIS
LIN {X 76.696,Y 144.867,Z 58.000,A 180.000,B 0.000,C 180.000} C_DIS
LIN {X 76.874,Y 144.920,Z 58.000,A 180.000,B 0.000,C 180.000} C_DIS
LIN {X 77.053,Y 144.960,Z 58.000,A 180.000,B 0.000,C 180.000} C_DIS
LIN {X 77.232,Y 144.986,Z 58.000,A 180.000,B 0.000,C 180.000} C_DIS
LIN {X 77.233,Y 144.986,Z 58.000,A 180.000,B 0.000,C 180.000} C_DIS
LIN {X 77.411,Y 144.998,Z 58.000,A 180.000,B 0.000,C 180.000} C_DIS
LIN {X 77.589,Y 144.998,Z 58.000,A 180.000,B 0.000,C 180.000} C_DIS
LIN {X 77.767,Y 144.986,Z 58.000,A 180.000,B 0.000,C 180.000} C_DIS
LIN {X 77.768,Y 144.986,Z 58.000,A 180.000,B 0.000,C 180.000} C_DIS
LIN {X 77.947,Y 144.960,Z 58.000,A 180.000,B 0.000,C 180.000} C_DIS
LIN {X 78.126,Y 144.920,Z 58.000,A 180.000,B 0.000,C 180.000} C_DIS
LIN {X 78.304,Y 144.867,Z 58.000,A 180.000,B 0.000,C 180.000} C_DIS
LIN {X 78.463,Y 144.807,Z 58.000,A 180.000,B 0.000,C 180.000} C_DIS
LIN {X 78.483,Y 144.799,Z 58.000,A 180.000,B 0.000,C 180.000} C_DIS
LIN {X 78.662,Y 144.714,Z 58.000,A 180.000,B 0.000,C 180.000} C_DIS
LIN {X 78.812,Y 144.628,Z 58.000,A 180.000,B 0.000,C 180.000} C_DIS
LIN {X 78.841,Y 144.610,Z 58.000,A 180.000,B 0.000,C 180.000} C_DIS
LIN {X 79.020,Y 144.485,Z 58.000,A 180.000,B 0.000,C 180.000} C_DIS
LIN {X 79.065,Y 144.449,Z 58.000,A 180.000,B 0.000,C 180.000} C_DIS
LIN {X 79.198,Y 144.335,Z 58.000,A 180.000,B 0.000,C 180.000} C_DIS
LIN {X 79.265,Y 144.271,Z 58.000,A 180.000,B 0.000,C 180.000} C_DIS
LIN {X 144.271,Y 79.265,Z 58.000,A 180.000,B 0.000,C 180.000} C_DIS
LIN {X 144.335,Y 79.198,Z 58.000,A 180.000,B 0.000,C 180.000} C_DIS
LIN {X 144.449,Y 79.065,Z 58.000,A 180.000,B 0.000,C 180.000} C_DIS
LIN {X 144.485,Y 79.020,Z 58.000,A 180.000,B 0.000,C 180.000} C_DIS
LIN {X 144.610,Y 78.841,Z 58.000,A 180.000,B 0.000,C 180.000} C_DIS
LIN {X 144.628,Y 78.812,Z 58.000,A 180.000,B 0.000,C 180.000} C_DIS
LIN {X 144.714,Y 78.662,Z 58.000,A 180.000,B 0.000,C 180.000} C_DIS
LIN {X 144.799,Y 78.483,Z 58.000,A 180.000,B 0.000,C 180.000} C_DIS
LIN {X 144.807,Y 78.463,Z 58.000,A 180.000,B 0.000,C 180.000} C_DIS
LIN {X 144.867,Y 78.304,Z 58.000,A 180.000,B 0.000,C 180.000} C_DIS
LIN {X 144.920,Y 78.126,Z 58.000,A 180.000,B 0.000,C 180.000} C_DIS
LIN {X 144.960,Y 77.947,Z 58.000,A 180.000,B 0.000,C 180.000} C_DIS
LIN {X 144.986,Y 77.768,Z 58.000,A 180.000,B 0.000,C 180.000} C_DIS
LIN {X 144.986,Y 77.767,Z 58.000,A 180.000,B 0.000,C 180.000} C_DIS
LIN {X 144.998,Y 77.589,Z 58.000,A 180.000,B 0.000,C 180.000} C_DIS
LIN {X 144.998,Y 77.411,Z 58.000,A 180.000,B 0.000,C 180.000} C_DIS
LIN {X 144.986,Y 77.233,Z 58.000,A 180.000,B 0.000,C 180.000} C_DIS
LIN {X 144.986,Y 77.232,Z 58.000,A 180.000,B 0.000,C 180.000} C_DIS
LIN {X 144.960,Y 77.053,Z 58.000,A 180.000,B 0.000,C 180.000} C_DIS
LIN {X 144.920,Y 76.874,Z 58.000,A 180.000,B 0.000,C 180.000} C_DIS
LIN {X 144.867,Y 76.696,Z 58.000,A 180.000,B 0.000,C 180.000} C_DIS
LIN {X 144.807,Y 76.537,Z 58.000,A 180.000,B 0.000,C 180.000} C_DIS
LIN {X 144.799,Y 76.517,Z 58.000,A 180.000,B 0.000,C 180.000} C_DIS
LIN {X 144.714,Y 76.338,Z 58.000,A 180.000,B 0.000,C 180.000} C_DIS
LIN {X 144.628,Y 76.188,Z 58.000,A 180.000,B 0.000,C 180.000} C_DIS
LIN {X 144.610,Y 76.159,Z 58.000,A 180.000,B 0.000,C 180.000} C_DIS
LIN {X 144.485,Y 75.980,Z 58.000,A 180.000,B 0.000,C 180.000} C_DIS
LIN {X 144.449,Y 75.935,Z 58.000,A 180.000,B 0.000,C 180.000} C_DIS
LIN {X 144.335,Y 75.802,Z 58.000,A 180.000,B 0.000,C 180.000} C_DIS
LIN {X 144.271,Y 75.735,Z 58.000,A 180.000,B 0.000,C 180.000} C_DIS
LIN {X 109.686,Y 41.150,Z 58.000,A 180.000,B 0.000,C 180.000} C_DIS
LIN {X 79.265,Y 10.729,Z 58.000,A 180.000,B 0.000,C 180.000} C_DIS
LIN {X 79.198,Y 10.665,Z 58.000,A 180.000,B 0.000,C 180.000} C_DIS
LIN {X 79.065,Y 10.551,Z 58.000,A 180.000,B 0.000,C 180.000} C_DIS
LIN {X 79.020,Y 10.515,Z 58.000,A 180.000,B 0.000,C 180.000} C_DIS
LIN {X 78.841,Y 10.390,Z 58.000,A 180.000,B 0.000,C 180.000} C_DIS
LIN {X 78.812,Y 10.372,Z 58.000,A 180.000,B 0.000,C 180.000} C_DIS
LIN {X 78.662,Y 10.286,Z 58.000,A 180.000,B 0.000,C 180.000} C_DIS
LIN {X 78.483,Y 10.201,Z 58.000,A 180.000,B 0.000,C 180.000} C_DIS
LIN {X 78.463,Y 10.193,Z 58.000,A 180.000,B 0.000,C 180.000} C_DIS
LIN {X 78.304,Y 10.133,Z 58.000,A 180.000,B 0.000,C 180.000} C_DIS
LIN {X 78.126,Y 10.080,Z 58.000,A 180.000,B 0.000,C 180.000} C_DIS
LIN {X 77.947,Y 10.040,Z 58.000,A 180.000,B 0.000,C 180.000} C_DIS
LIN {X 77.768,Y 10.014,Z 58.000,A 180.000,B 0.000,C 180.000} C_DIS
LIN {X 77.767,Y 10.014,Z 58.000,A 180.000,B 0.000,C 180.000} C_DIS
LIN {X 77.589,Y 10.002,Z 58.000,A 180.000,B 0.000,C 180.000} C_DIS
LIN {X 77.411,Y 10.002,Z 58.000,A 180.000,B 0.000,C 180.000} C_DIS
LIN {X 77.233,Y 10.014,Z 58.000,A 180.000,B 0.000,C 180.000} C_DIS
LIN {X 77.232,Y 10.014,Z 58.000,A 180.000,B 0.000,C 180.000} C_DIS
LIN {X 77.053,Y 10.040,Z 58.000,A 180.000,B 0.000,C 180.000} C_DIS
LIN {X 76.874,Y 10.080,Z 58.000,A 180.000,B 0.000,C 180.000} C_DIS
LIN {X 76.696,Y 10.133,Z 58.000,A 180.000,B 0.000,C 180.000} C_DIS
LIN {X 76.537,Y 10.193,Z 58.000,A 180.000,B 0.000,C 180.000} C_DIS
LIN {X 76.517,Y 10.201,Z 58.000,A 180.000,B 0.000,C 180.000} C_DIS
LIN {X 76.338,Y 10.286,Z 58.000,A 180.000,B 0.000,C 180.000} C_DIS
LIN {X 76.188,Y 10.372,Z 58.000,A 180.000,B 0.000,C 180.000} C_DIS
LIN {X 76.159,Y 10.390,Z 58.000,A 180.000,B 0.000,C 180.000} C_DIS
LIN {X 75.980,Y 10.515,Z 58.000,A 180.000,B 0.000,C 180.000} C_DIS
LIN {X 75.935,Y 10.551,Z 58.000,A 180.000,B 0.000,C 180.000} C_DIS
LIN {X 75.802,Y 10.665,Z 58.000,A 180.000,B 0.000,C 180.000} C_DIS
LIN {X 75.735,Y 10.729,Z 58.000,A 180.000,B 0.000,C 180.000} C_DIS
LIN {X 33.829,Y 52.636,Z 58.000,A 180.000,B 0.000,C 180.000} C_DIS
; Link Move Starts
LIN {X 33.606,Y 52.858,Z 58.000,A 180.000,B 0.000,C 180.000} C_DIS
LIN {X 33.383,Y 53.081,Z 57.999,A 180.000,B 0.000,C 180.000} C_DIS
LIN {X 33.161,Y 53.304,Z 57.998,A 180.000,B 0.000,C 180.000} C_DIS
LIN {X 32.938,Y 53.526,Z 57.996,A 180.000,B 0.000,C 180.000} C_DIS
LIN {X 32.715,Y 53.749,Z 57.994,A 180.000,B 0.000,C 180.000} C_DIS
LIN {X 32.493,Y 53.972,Z 57.991,A 180.000,B 0.000,C 180.000} C_DIS
LIN {X 32.270,Y 54.195,Z 57.988,A 180.000,B 0.000,C 180.000} C_DIS
LIN {X 32.047,Y 54.417,Z 57.985,A 180.000,B 0.000,C 180.000} C_DIS
LIN {X 31.824,Y 54.640,Z 57.981,A 180.000,B 0.000,C 180.000} C_DIS
LIN {X 31.602,Y 54.863,Z 57.977,A 180.000,B 0.000,C 180.000} C_DIS
LIN {X 31.379,Y 55.086,Z 57.972,A 180.000,B 0.000,C 180.000} C_DIS
LIN {X 31.267,Y 55.197,Z 57.969,A 180.000,B 0.000,C 180.000} C_DIS
LIN {X 31.156,Y 55.308,Z 57.967,A 180.000,B 0.000,C 180.000} C_DIS
LIN {X 31.045,Y 55.420,Z 57.964,A 180.000,B 0.000,C 180.000} C_DIS
LIN {X 30.933,Y 55.531,Z 57.961,A 180.000,B 0.000,C 180.000} C_DIS
LIN {X 30.822,Y 55.642,Z 57.959,A 180.000,B 0.000,C 180.000} C_DIS
LIN {X 30.711,Y 55.754,Z 57.956,A 180.000,B 0.000,C 180.000} C_DIS
LIN {X 30.599,Y 55.865,Z 57.952,A 180.000,B 0.000,C 180.000} C_DIS
LIN {X 30.488,Y 55.977,Z 57.949,A 180.000,B 0.000,C 180.000} C_DIS
LIN {X 30.377,Y 56.088,Z 57.946,A 180.000,B 0.000,C 180.000} C_DIS
LIN {X 30.265,Y 56.199,Z 57.943,A 180.000,B 0.000,C 180.000} C_DIS
LIN {X 30.154,Y 56.311,Z 57.939,A 180.000,B 0.000,C 180.000} C_DIS
LIN {X 30.042,Y 56.422,Z 57.936,A 180.000,B 0.000,C 180.000} C_DIS
LIN {X 29.931,Y 56.533,Z 57.932,A 180.000,B 0.000,C 180.000} C_DIS
LIN {X 29.820,Y 56.645,Z 57.928,A 180.000,B 0.000,C 180.000} C_DIS
LIN {X 29.708,Y 56.756,Z 57.925,A 180.000,B 0.000,C 180.000} C_DIS
LIN {X 29.597,Y 56.868,Z 57.921,A 180.000,B 0.000,C 180.000} C_DIS
LIN {X 29.486,Y 56.979,Z 57.917,A 180.000,B 0.000,C 180.000} C_DIS
LIN {X 29.374,Y 57.090,Z 57.913,A 180.000,B 0.000,C 180.000} C_DIS
LIN {X 29.263,Y 57.202,Z 57.909,A 180.000,B 0.000,C 180.000} C_DIS
LIN {X 29.151,Y 57.313,Z 57.905,A 180.000,B 0.000,C 180.000} C_DIS
LIN {X 29.040,Y 57.424,Z 57.900,A 180.000,B 0.000,C 180.000} C_DIS
LIN {X 28.929,Y 57.536,Z 57.896,A 180.000,B 0.000,C 180.000} C_DIS
LIN {X 28.817,Y 57.647,Z 57.892,A 180.000,B 0.000,C 180.000} C_DIS
LIN {X 28.706,Y 57.758,Z 57.887,A 180.000,B 0.000,C 180.000} C_DIS
LIN {X 28.595,Y 57.870,Z 57.883,A 180.000,B 0.000,C 180.000} C_DIS
LIN {X 28.483,Y 57.981,Z 57.878,A 180.000,B 0.000,C 180.000} C_DIS
LIN {X 28.372,Y 58.093,Z 57.873,A 180.000,B 0.000,C 180.000} C_DIS
LIN {X 28.260,Y 58.204,Z 57.869,A 180.000,B 0.000,C 180.000} C_DIS
LIN {X 28.149,Y 58.315,Z 57.864,A 180.000,B 0.000,C 180.000} C_DIS
LIN {X 28.038,Y 58.427,Z 57.859,A 180.000,B 0.000,C 180.000} C_DIS
LIN {X 27.926,Y 58.538,Z 57.854,A 180.000,B 0.000,C 180.000} C_DIS
LIN {X 27.871,Y 58.594,Z 57.851,A 180.000,B 0.000,C 180.000} C_DIS
LIN {X 27.815,Y 58.649,Z 57.849,A 180.000,B 0.000,C 180.000} C_DIS
LIN {X 27.759,Y 58.705,Z 57.846,A 180.000,B 0.000,C 180.000} C_DIS
LIN {X 27.704,Y 58.761,Z 57.844,A 180.000,B 0.000,C 180.000} C_DIS
LIN {X 27.648,Y 58.817,Z 57.841,A 180.000,B 0.000,C 180.000} C_DIS
LIN {X 27.592,Y 58.872,Z 57.839,A 180.000,B 0.000,C 180.000} C_DIS
LIN {X 27.537,Y 58.928,Z 57.836,A 180.000,B 0.000,C 180.000} C_DIS
LIN {X 27.425,Y 59.039,Z 57.831,A 180.000,B 0.000,C 180.000} C_DIS
LIN {X 27.314,Y 59.151,Z 57.825,A 180.000,B 0.000,C 180.000} C_DIS
LIN {X 27.202,Y 59.262,Z 57.820,A 180.000,B 0.000,C 180.000} C_DIS
LIN {X 27.091,Y 59.373,Z 57.815,A 180.000,B 0.000,C 180.000} C_DIS
LIN {X 26.980,Y 59.485,Z 57.809,A 180.000,B 0.000,C 180.000} C_DIS
LIN {X 26.924,Y 59.540,Z 57.806,A 180.000,B 0.000,C 180.000} C_DIS
LIN {X 26.813,Y 59.652,Z 57.801,A 180.000,B 0.000,C 180.000} C_DIS
LIN {X 26.646,Y 59.819,Z 57.793,A 180.000,B 0.000,C 180.000} C_DIS
LIN {X 26.534,Y 59.930,Z 57.787,A 180.000,B 0.000,C 180.000} C_DIS
LIN {X 26.479,Y 59.986,Z 57.785,A 180.000,B 0.000,C 180.000} C_DIS
LIN {X 26.367,Y 60.097,Z 57.779,A 180.000,B 0.000,C 180.000} C_DIS
LIN {X 26.200,Y 60.264,Z 57.771,A 180.000,B 0.000,C 180.000} C_DIS
LIN {X 26.089,Y 60.376,Z 57.765,A 180.000,B 0.000,C 180.000} C_DIS
LIN {X 26.033,Y 60.431,Z 57.763,A 180.000,B 0.000,C 180.000} C_DIS
LIN {X 25.922,Y 60.543,Z 57.757,A 180.000,B 0.000,C 180.000} C_DIS
LIN {X 25.755,Y 60.710,Z 57.749,A 180.000,B 0.000,C 180.000} C_DIS
LIN {X 25.643,Y 60.821,Z 57.743,A 180.000,B 0.000,C 180.000} C_DIS
LIN {X 25.588,Y 60.877,Z 57.741,A 180.000,B 0.000,C 180.000} C_DIS
LIN {X 25.476,Y 60.988,Z 57.735,A 180.000,B 0.000,C 180.000} C_DIS
LIN {X 25.309,Y 61.155,Z 57.727,A 180.000,B 0.000,C 180.000} C_DIS
LIN {X 25.198,Y 61.267,Z 57.721,A 180.000,B 0.000,C 180.000} C_DIS
LIN {X 25.142,Y 61.322,Z 57.719,A 180.000,B 0.000,C 180.000} C_DIS
LIN {X 25.031,Y 61.434,Z 57.713,A 180.000,B 0.000,C 180.000} C_DIS
LIN {X 24.697,Y 61.768,Z 57.697,A 180.000,B 0.000,C 180.000} C_DIS
LIN {X 24.585,Y 61.879,Z 57.691,A 180.000,B 0.000,C 180.000} C_DIS
LIN {X 24.251,Y 62.213,Z 57.675,A 180.000,B 0.000,C 180.000} C_DIS
LIN {X 24.140,Y 62.325,Z 57.669,A 180.000,B 0.000,C 180.000} C_DIS
LIN {X 23.750,Y 62.714,Z 57.650,A 180.000,B 0.000,C 180.000} C_DIS
LIN {X 23.416,Y 63.049,Z 57.633,A 180.000,B 0.000,C 180.000} C_DIS
LIN {X 23.305,Y 63.160,Z 57.628,A 180.000,B 0.000,C 180.000} C_DIS
LIN {X 22.970,Y 63.494,Z 57.611,A 180.000,B 0.000,C 180.000} C_DIS
LIN {X 22.859,Y 63.605,Z 57.606,A 180.000,B 0.000,C 180.000} C_DIS
LIN {X 22.302,Y 64.162,Z 57.578,A 180.000,B 0.000,C 180.000} C_DIS
LIN {X 22.024,Y 64.441,Z 57.565,A 180.000,B 0.000,C 180.000} C_DIS
LIN {X 21.690,Y 64.775,Z 57.548,A 180.000,B 0.000,C 180.000} C_DIS
LIN {X 20.409,Y 66.055,Z 57.485,A 180.000,B 0.000,C 180.000} C_DIS
LIN {X 18.293,Y 68.171,Z 57.380,A 180.000,B 0.000,C 180.000} C_DIS
LIN {X 18.182,Y 68.283,Z 57.375,A 180.000,B 0.000,C 180.000} C_DIS
LIN {X 17.847,Y 68.617,Z 57.358,A 180.000,B 0.000,C 180.000} C_DIS
LIN {X 17.736,Y 68.728,Z 57.353,A 180.000,B 0.000,C 180.000} C_DIS
LIN {X 17.402,Y 69.062,Z 57.336,A 180.000,B 0.000,C 180.000} C_DIS
LIN {X 17.346,Y 69.118,Z 57.334,A 180.000,B 0.000,C 180.000} C_DIS
LIN {X 17.235,Y 69.229,Z 57.328,A 180.000,B 0.000,C 180.000} C_DIS
LIN {X 16.901,Y 69.564,Z 57.312,A 180.000,B 0.000,C 180.000} C_DIS
LIN {X 16.789,Y 69.675,Z 57.306,A 180.000,B 0.000,C 180.000} C_DIS
LIN {X 16.455,Y 70.009,Z 57.290,A 180.000,B 0.000,C 180.000} C_DIS
LIN {X 16.344,Y 70.120,Z 57.284,A 180.000,B 0.000,C 180.000} C_DIS
LIN {X 16.177,Y 70.287,Z 57.276,A 180.000,B 0.000,C 180.000} C_DIS
LIN {X 16.066,Y 70.399,Z 57.270,A 180.000,B 0.000,C 180.000} C_DIS
LIN {X 16.010,Y 70.455,Z 57.268,A 180.000,B 0.000,C 180.000} C_DIS
LIN {X 15.899,Y 70.566,Z 57.262,A 180.000,B 0.000,C 180.000} C_DIS
LIN {X 15.731,Y 70.733,Z 57.254,A 180.000,B 0.000,C 180.000} C_DIS
LIN {X 15.620,Y 70.844,Z 57.248,A 180.000,B 0.000,C 180.000} C_DIS
LIN {X 15.564,Y 70.900,Z 57.246,A 180.000,B 0.000,C 180.000} C_DIS
LIN {X 15.453,Y 71.011,Z 57.240,A 180.000,B 0.000,C 180.000} C_DIS
LIN {X 15.286,Y 71.178,Z 57.232,A 180.000,B 0.000,C 180.000} C_DIS
LIN {X 15.175,Y 71.290,Z 57.226,A 180.000,B 0.000,C 180.000} C_DIS
LIN {X 15.119,Y 71.346,Z 57.224,A 180.000,B 0.000,C 180.000} C_DIS
LIN {X 15.008,Y 71.457,Z 57.218,A 180.000,B 0.000,C 180.000} C_DIS
LIN {X 14.841,Y 71.624,Z 57.210,A 180.000,B 0.000,C 180.000} C_DIS
LIN {X 14.729,Y 71.735,Z 57.204,A 180.000,B 0.000,C 180.000} C_DIS
LIN {X 14.673,Y 71.791,Z 57.202,A 180.000,B 0.000,C 180.000} C_DIS
LIN {X 14.562,Y 71.902,Z 57.196,A 180.000,B 0.000,C 180.000} C_DIS
LIN {X 14.451,Y 72.014,Z 57.191,A 180.000,B 0.000,C 180.000} C_DIS
LIN {X 14.339,Y 72.125,Z 57.185,A 180.000,B 0.000,C 180.000} C_DIS
LIN {X 14.228,Y 72.236,Z 57.180,A 180.000,B 0.000,C 180.000} C_DIS
LIN {X 14.117,Y 72.348,Z 57.174,A 180.000,B 0.000,C 180.000} C_DIS
LIN {X 14.005,Y 72.459,Z 57.169,A 180.000,B 0.000,C 180.000} C_DIS
LIN {X 13.894,Y 72.571,Z 57.164,A 180.000,B 0.000,C 180.000} C_DIS
LIN {X 13.838,Y 72.626,Z 57.161,A 180.000,B 0.000,C 180.000} C_DIS
LIN {X 13.783,Y 72.682,Z 57.159,A 180.000,B 0.000,C 180.000} C_DIS
LIN {X 13.727,Y 72.738,Z 57.156,A 180.000,B 0.000,C 180.000} C_DIS
LIN {X 13.671,Y 72.793,Z 57.154,A 180.000,B 0.000,C 180.000} C_DIS
LIN {X 13.615,Y 72.849,Z 57.151,A 180.000,B 0.000,C 180.000} C_DIS
LIN {X 13.560,Y 72.905,Z 57.148,A 180.000,B 0.000,C 180.000} C_DIS
LIN {X 13.448,Y 73.016,Z 57.143,A 180.000,B 0.000,C 180.000} C_DIS
LIN {X 13.337,Y 73.127,Z 57.139,A 180.000,B 0.000,C 180.000} C_DIS
LIN {X 13.226,Y 73.239,Z 57.134,A 180.000,B 0.000,C 180.000} C_DIS
LIN {X 13.114,Y 73.350,Z 57.129,A 180.000,B 0.000,C 180.000} C_DIS
LIN {X 13.003,Y 73.462,Z 57.124,A 180.000,B 0.000,C 180.000} C_DIS
LIN {X 12.892,Y 73.573,Z 57.120,A 180.000,B 0.000,C 180.000} C_DIS
LIN {X 12.780,Y 73.684,Z 57.115,A 180.000,B 0.000,C 180.000} C_DIS
LIN {X 12.669,Y 73.796,Z 57.110,A 180.000,B 0.000,C 180.000} C_DIS
LIN {X 12.557,Y 73.907,Z 57.106,A 180.000,B 0.000,C 180.000} C_DIS
LIN {X 12.446,Y 74.018,Z 57.102,A 180.000,B 0.000,C 180.000} C_DIS
LIN {X 12.335,Y 74.130,Z 57.097,A 180.000,B 0.000,C 180.000} C_DIS
LIN {X 12.223,Y 74.241,Z 57.093,A 180.000,B 0.000,C 180.000} C_DIS
LIN {X 12.112,Y 74.352,Z 57.089,A 180.000,B 0.000,C 180.000} C_DIS
LIN {X 12.001,Y 74.464,Z 57.085,A 180.000,B 0.000,C 180.000} C_DIS
LIN {X 11.889,Y 74.575,Z 57.081,A 180.000,B 0.000,C 180.000} C_DIS
LIN {X 11.778,Y 74.687,Z 57.077,A 180.000,B 0.000,C 180.000} C_DIS
LIN {X 11.667,Y 74.798,Z 57.073,A 180.000,B 0.000,C 180.000} C_DIS
LIN {X 11.555,Y 74.909,Z 57.070,A 180.000,B 0.000,C 180.000} C_DIS
LIN {X 11.444,Y 75.021,Z 57.066,A 180.000,B 0.000,C 180.000} C_DIS
LIN {X 11.332,Y 75.132,Z 57.062,A 180.000,B 0.000,C 180.000} C_DIS
LIN {X 11.221,Y 75.243,Z 57.059,A 180.000,B 0.000,C 180.000} C_DIS
LIN {X 11.110,Y 75.355,Z 57.056,A 180.000,B 0.000,C 180.000} C_DIS
LIN {X 10.998,Y 75.466,Z 57.052,A 180.000,B 0.000,C 180.000} C_DIS
LIN {X 10.887,Y 75.578,Z 57.049,A 180.000,B 0.000,C 180.000} C_DIS
LIN {X 10.776,Y 75.689,Z 57.046,A 180.000,B 0.000,C 180.000} C_DIS
LIN {X 10.666,Y 75.802,Z 57.043,A 180.000,B 0.000,C 180.000} C_DIS
LIN {X 10.562,Y 75.920,Z 57.040,A 180.000,B 0.000,C 180.000} C_DIS
LIN {X 10.467,Y 76.046,Z 57.037,A 180.000,B 0.000,C 180.000} C_DIS
LIN {X 10.379,Y 76.177,Z 57.034,A 180.000,B 0.000,C 180.000} C_DIS
LIN {X 10.300,Y 76.313,Z 57.032,A 180.000,B 0.000,C 180.000} C_DIS
LIN {X 10.230,Y 76.454,Z 57.029,A 180.000,B 0.000,C 180.000} C_DIS
LIN {X 10.168,Y 76.599,Z 57.027,A 180.000,B 0.000,C 180.000} C_DIS
LIN {X 10.116,Y 76.747,Z 57.024,A 180.000,B 0.000,C 180.000} C_DIS
LIN {X 10.073,Y 76.899,Z 57.022,A 180.000,B 0.000,C 180.000} C_DIS
LIN {X 10.040,Y 77.053,Z 57.020,A 180.000,B 0.000,C 180.000} C_DIS
LIN {X 10.017,Y 77.209,Z 57.018,A 180.000,B 0.000,C 180.000} C_DIS
LIN {X 10.004,Y 77.366,Z 57.016,A 180.000,B 0.000,C 180.000} C_DIS
LIN {X 10.000,Y 77.523,Z 57.014,A 180.000,B 0.000,C 180.000} C_DIS
LIN {X 10.007,Y 77.680,Z 57.012,A 180.000,B 0.000,C 180.000} C_DIS
LIN {X 10.023,Y 77.837,Z 57.011,A 180.000,B 0.000,C 180.000} C_DIS
LIN {X 10.049,Y 77.992,Z 57.009,A 180.000,B 0.000,C 180.000} C_DIS
LIN {X 10.085,Y 78.146,Z 57.008,A 180.000,B 0.000,C 180.000} C_DIS
LIN {X 10.130,Y 78.297,Z 57.007,A 180.000,B 0.000,C 180.000} C_DIS
LIN {X 10.185,Y 78.444,Z 57.005,A 180.000,B 0.000,C 180.000} C_DIS
LIN {X 10.249,Y 78.588,Z 57.004,A 180.000,B 0.000,C 180.000} C_DIS
LIN {X 10.322,Y 78.728,Z 57.003,A 180.000,B 0.000,C 180.000} C_DIS
LIN {X 10.404,Y 78.862,Z 57.003,A 180.000,B 0.000,C 180.000} C_DIS
LIN {X 10.494,Y 78.992,Z 57.002,A 180.000,B 0.000,C 180.000} C_DIS
LIN {X 10.592,Y 79.115,Z 57.001,A 180.000,B 0.000,C 180.000} C_DIS
LIN {X 10.697,Y 79.232,Z 57.001,A 180.000,B 0.000,C 180.000} C_DIS
LIN {X 10.920,Y 79.455,Z 57.000,A 180.000,B 0.000,C 180.000} C_DIS
LIN {X 11.083,Y 79.618,Z 57.000,A 180.000,B 0.000,C 180.000} C_DIS
; Cutting Move Starts
LIN {X 75.735,Y 144.271,Z 57.000,A 180.000,B 0.000,C 180.000} C_DIS
LIN {X 75.802,Y 144.335,Z 57.000,A 180.000,B 0.000,C 180.000} C_DIS
LIN {X 75.935,Y 144.449,Z 57.000,A 180.000,B 0.000,C 180.000} C_DIS
LIN {X 75.980,Y 144.485,Z 57.000,A 180.000,B 0.000,C 180.000} C_DIS
LIN {X 76.159,Y 144.610,Z 57.000,A 180.000,B 0.000,C 180.000} C_DIS
LIN {X 76.188,Y 144.628,Z 57.000,A 180.000,B 0.000,C 180.000} C_DIS
LIN {X 76.338,Y 144.714,Z 57.000,A 180.000,B 0.000,C 180.000} C_DIS
LIN {X 76.517,Y 144.799,Z 57.000,A 180.000,B 0.000,C 180.000} C_DIS
LIN {X 76.537,Y 144.807,Z 57.000,A 180.000,B 0.000,C 180.000} C_DIS
LIN {X 76.696,Y 144.867,Z 57.000,A 180.000,B 0.000,C 180.000} C_DIS
LIN {X 76.874,Y 144.920,Z 57.000,A 180.000,B 0.000,C 180.000} C_DIS
LIN {X 77.053,Y 144.960,Z 57.000,A 180.000,B 0.000,C 180.000} C_DIS
LIN {X 77.232,Y 144.986,Z 57.000,A 180.000,B 0.000,C 180.000} C_DIS
LIN {X 77.233,Y 144.986,Z 57.000,A 180.000,B 0.000,C 180.000} C_DIS
LIN {X 77.411,Y 144.998,Z 57.000,A 180.000,B 0.000,C 180.000} C_DIS
LIN {X 77.589,Y 144.998,Z 57.000,A 180.000,B 0.000,C 180.000} C_DIS
LIN {X 77.767,Y 144.986,Z 57.000,A 180.000,B 0.000,C 180.000} C_DIS
LIN {X 77.768,Y 144.986,Z 57.000,A 180.000,B 0.000,C 180.000} C_DIS
LIN {X 77.947,Y 144.960,Z 57.000,A 180.000,B 0.000,C 180.000} C_DIS
LIN {X 78.126,Y 144.920,Z 57.000,A 180.000,B 0.000,C 180.000} C_DIS
LIN {X 78.304,Y 144.867,Z 57.000,A 180.000,B 0.000,C 180.000} C_DIS
LIN {X 78.463,Y 144.807,Z 57.000,A 180.000,B 0.000,C 180.000} C_DIS
LIN {X 78.483,Y 144.799,Z 57.000,A 180.000,B 0.000,C 180.000} C_DIS
LIN {X 78.662,Y 144.714,Z 57.000,A 180.000,B 0.000,C 180.000} C_DIS
LIN {X 78.812,Y 144.628,Z 57.000,A 180.000,B 0.000,C 180.000} C_DIS
LIN {X 78.841,Y 144.610,Z 57.000,A 180.000,B 0.000,C 180.000} C_DIS
LIN {X 79.020,Y 144.485,Z 57.000,A 180.000,B 0.000,C 180.000} C_DIS
LIN {X 79.065,Y 144.449,Z 57.000,A 180.000,B 0.000,C 180.000} C_DIS
LIN {X 79.198,Y 144.335,Z 57.000,A 180.000,B 0.000,C 180.000} C_DIS
LIN {X 79.265,Y 144.271,Z 57.000,A 180.000,B 0.000,C 180.000} C_DIS
LIN {X 144.271,Y 79.265,Z 57.000,A 180.000,B 0.000,C 180.000} C_DIS
LIN {X 144.335,Y 79.198,Z 57.000,A 180.000,B 0.000,C 180.000} C_DIS
LIN {X 144.449,Y 79.065,Z 57.000,A 180.000,B 0.000,C 180.000} C_DIS
LIN {X 144.485,Y 79.020,Z 57.000,A 180.000,B 0.000,C 180.000} C_DIS
LIN {X 144.610,Y 78.841,Z 57.000,A 180.000,B 0.000,C 180.000} C_DIS
LIN {X 144.628,Y 78.812,Z 57.000,A 180.000,B 0.000,C 180.000} C_DIS
LIN {X 144.714,Y 78.662,Z 57.000,A 180.000,B 0.000,C 180.000} C_DIS
LIN {X 144.799,Y 78.483,Z 57.000,A 180.000,B 0.000,C 180.000} C_DIS
LIN {X 144.807,Y 78.463,Z 57.000,A 180.000,B 0.000,C 180.000} C_DIS
LIN {X 144.867,Y 78.304,Z 57.000,A 180.000,B 0.000,C 180.000} C_DIS
LIN {X 144.920,Y 78.126,Z 57.000,A 180.000,B 0.000,C 180.000} C_DIS
LIN {X 144.960,Y 77.947,Z 57.000,A 180.000,B 0.000,C 180.000} C_DIS
LIN {X 144.986,Y 77.768,Z 57.000,A 180.000,B 0.000,C 180.000} C_DIS
LIN {X 144.986,Y 77.767,Z 57.000,A 180.000,B 0.000,C 180.000} C_DIS
LIN {X 144.998,Y 77.589,Z 57.000,A 180.000,B 0.000,C 180.000} C_DIS
LIN {X 144.998,Y 77.411,Z 57.000,A 180.000,B 0.000,C 180.000} C_DIS
LIN {X 144.986,Y 77.233,Z 57.000,A 180.000,B 0.000,C 180.000} C_DIS
LIN {X 144.986,Y 77.232,Z 57.000,A 180.000,B 0.000,C 180.000} C_DIS
LIN {X 144.960,Y 77.053,Z 57.000,A 180.000,B 0.000,C 180.000} C_DIS
LIN {X 144.920,Y 76.874,Z 57.000,A 180.000,B 0.000,C 180.000} C_DIS
LIN {X 144.867,Y 76.696,Z 57.000,A 180.000,B 0.000,C 180.000} C_DIS
LIN {X 144.807,Y 76.537,Z 57.000,A 180.000,B 0.000,C 180.000} C_DIS
LIN {X 144.799,Y 76.517,Z 57.000,A 180.000,B 0.000,C 180.000} C_DIS
LIN {X 144.714,Y 76.338,Z 57.000,A 180.000,B 0.000,C 180.000} C_DIS
LIN {X 144.628,Y 76.188,Z 57.000,A 180.000,B 0.000,C 180.000} C_DIS
LIN {X 144.610,Y 76.159,Z 57.000,A 180.000,B 0.000,C 180.000} C_DIS
LIN {X 144.485,Y 75.980,Z 57.000,A 180.000,B 0.000,C 180.000} C_DIS
LIN {X 144.449,Y 75.935,Z 57.000,A 180.000,B 0.000,C 180.000} C_DIS
LIN {X 144.335,Y 75.802,Z 57.000,A 180.000,B 0.000,C 180.000} C_DIS
LIN {X 144.271,Y 75.735,Z 57.000,A 180.000,B 0.000,C 180.000} C_DIS
LIN {X 109.686,Y 41.150,Z 57.000,A 180.000,B 0.000,C 180.000} C_DIS
LIN {X 79.265,Y 10.729,Z 57.000,A 180.000,B 0.000,C 180.000} C_DIS
LIN {X 79.198,Y 10.665,Z 57.000,A 180.000,B 0.000,C 180.000} C_DIS
LIN {X 79.065,Y 10.551,Z 57.000,A 180.000,B 0.000,C 180.000} C_DIS
LIN {X 79.020,Y 10.515,Z 57.000,A 180.000,B 0.000,C 180.000} C_DIS
LIN {X 78.841,Y 10.390,Z 57.000,A 180.000,B 0.000,C 180.000} C_DIS
LIN {X 78.812,Y 10.372,Z 57.000,A 180.000,B 0.000,C 180.000} C_DIS
LIN {X 78.662,Y 10.286,Z 57.000,A 180.000,B 0.000,C 180.000} C_DIS
LIN {X 78.483,Y 10.201,Z 57.000,A 180.000,B 0.000,C 180.000} C_DIS
LIN {X 78.463,Y 10.193,Z 57.000,A 180.000,B 0.000,C 180.000} C_DIS
LIN {X 78.304,Y 10.133,Z 57.000,A 180.000,B 0.000,C 180.000} C_DIS
LIN {X 78.126,Y 10.080,Z 57.000,A 180.000,B 0.000,C 180.000} C_DIS
LIN {X 77.947,Y 10.040,Z 57.000,A 180.000,B 0.000,C 180.000} C_DIS
LIN {X 77.768,Y 10.014,Z 57.000,A 180.000,B 0.000,C 180.000} C_DIS
LIN {X 77.767,Y 10.014,Z 57.000,A 180.000,B 0.000,C 180.000} C_DIS
LIN {X 77.589,Y 10.002,Z 57.000,A 180.000,B 0.000,C 180.000} C_DIS
LIN {X 77.411,Y 10.002,Z 57.000,A 180.000,B 0.000,C 180.000} C_DIS
LIN {X 77.233,Y 10.014,Z 57.000,A 180.000,B 0.000,C 180.000} C_DIS
LIN {X 77.232,Y 10.014,Z 57.000,A 180.000,B 0.000,C 180.000} C_DIS
LIN {X 77.053,Y 10.040,Z 57.000,A 180.000,B 0.000,C 180.000} C_DIS
LIN {X 76.874,Y 10.080,Z 57.000,A 180.000,B 0.000,C 180.000} C_DIS
LIN {X 76.696,Y 10.133,Z 57.000,A 180.000,B 0.000,C 180.000} C_DIS
LIN {X 76.537,Y 10.193,Z 57.000,A 180.000,B 0.000,C 180.000} C_DIS
LIN {X 76.517,Y 10.201,Z 57.000,A 180.000,B 0.000,C 180.000} C_DIS
LIN {X 76.338,Y 10.286,Z 57.000,A 180.000,B 0.000,C 180.000} C_DIS
LIN {X 76.188,Y 10.372,Z 57.000,A 180.000,B 0.000,C 180.000} C_DIS
LIN {X 76.159,Y 10.390,Z 57.000,A 180.000,B 0.000,C 180.000} C_DIS
LIN {X 75.980,Y 10.515,Z 57.000,A 180.000,B 0.000,C 180.000} C_DIS
LIN {X 75.935,Y 10.551,Z 57.000,A 180.000,B 0.000,C 180.000} C_DIS
LIN {X 75.802,Y 10.665,Z 57.000,A 180.000,B 0.000,C 180.000} C_DIS
LIN {X 75.735,Y 10.729,Z 57.000,A 180.000,B 0.000,C 180.000} C_DIS
LIN {X 33.829,Y 52.636,Z 57.000,A 180.000,B 0.000,C 180.000} C_DIS
LIN {X 10.729,Y 75.735,Z 57.000,A 180.000,B 0.000,C 180.000} C_DIS
LIN {X 10.665,Y 75.802,Z 57.000,A 180.000,B 0.000,C 180.000} C_DIS
LIN {X 10.551,Y 75.935,Z 57.000,A 180.000,B 0.000,C 180.000} C_DIS
LIN {X 10.515,Y 75.980,Z 57.000,A 180.000,B 0.000,C 180.000} C_DIS
LIN {X 10.390,Y 76.159,Z 57.000,A 180.000,B 0.000,C 180.000} C_DIS
LIN {X 10.372,Y 76.188,Z 57.000,A 180.000,B 0.000,C 180.000} C_DIS
LIN {X 10.286,Y 76.338,Z 57.000,A 180.000,B 0.000,C 180.000} C_DIS
LIN {X 10.201,Y 76.517,Z 57.000,A 180.000,B 0.000,C 180.000} C_DIS
LIN {X 10.193,Y 76.537,Z 57.000,A 180.000,B 0.000,C 180.000} C_DIS
LIN {X 10.133,Y 76.696,Z 57.000,A 180.000,B 0.000,C 180.000} C_DIS
LIN {X 10.080,Y 76.874,Z 57.000,A 180.000,B 0.000,C 180.000} C_DIS
LIN {X 10.040,Y 77.053,Z 57.000,A 180.000,B 0.000,C 180.000} C_DIS
LIN {X 10.014,Y 77.232,Z 57.000,A 180.000,B 0.000,C 180.000} C_DIS
LIN {X 10.014,Y 77.233,Z 57.000,A 180.000,B 0.000,C 180.000} C_DIS
LIN {X 10.002,Y 77.411,Z 57.000,A 180.000,B 0.000,C 180.000} C_DIS
LIN {X 10.002,Y 77.589,Z 57.000,A 180.000,B 0.000,C 180.000} C_DIS
LIN {X 10.014,Y 77.767,Z 57.000,A 180.000,B 0.000,C 180.000} C_DIS
LIN {X 10.014,Y 77.768,Z 57.000,A 180.000,B 0.000,C 180.000} C_DIS
LIN {X 10.040,Y 77.947,Z 57.000,A 180.000,B 0.000,C 180.000} C_DIS
LIN {X 10.080,Y 78.126,Z 57.000,A 180.000,B 0.000,C 180.000} C_DIS
LIN {X 10.133,Y 78.304,Z 57.000,A 180.000,B 0.000,C 180.000} C_DIS
LIN {X 10.193,Y 78.463,Z 57.000,A 180.000,B 0.000,C 180.000} C_DIS
LIN {X 10.201,Y 78.483,Z 57.000,A 180.000,B 0.000,C 180.000} C_DIS
LIN {X 10.286,Y 78.662,Z 57.000,A 180.000,B 0.000,C 180.000} C_DIS
LIN {X 10.372,Y 78.812,Z 57.000,A 180.000,B 0.000,C 180.000} C_DIS
LIN {X 10.390,Y 78.841,Z 57.000,A 180.000,B 0.000,C 180.000} C_DIS
LIN {X 10.515,Y 79.020,Z 57.000,A 180.000,B 0.000,C 180.000} C_DIS
LIN {X 10.551,Y 79.065,Z 57.000,A 180.000,B 0.000,C 180.000} C_DIS
LIN {X 10.665,Y 79.198,Z 57.000,A 180.000,B 0.000,C 180.000} C_DIS
LIN {X 10.729,Y 79.265,Z 57.000,A 180.000,B 0.000,C 180.000} C_DIS
LIN {X 11.083,Y 79.618,Z 57.000,A 180.000,B 0.000,C 180.000} C_DIS
; Lead Out Move Starts
LIN {X 11.222,Y 80.056,Z 57.000,A 180.000,B 0.000,C 180.000} C_DIS
LIN {X 10.945,Y 80.423,Z 57.000,A 180.000,B 0.000,C 180.000} C_DIS
LIN {X 10.120,Y 80.818,Z 57.000,A 180.000,B 0.000,C 180.000} C_DIS
LIN {X 9.801,Y 80.970,Z 57.146,A 180.000,B 0.000,C 180.000} C_DIS
LIN {X 9.669,Y 81.034,Z 57.500,A 180.000,B 0.000,C 180.000} C_DIS
; Rapid Move Starts
LIN {X 9.669,Y 81.034,Z 95.000,A 180.000,B 0.000,C 180.000} C_DIS
LIN {X 113.003,Y 39.300,Z 95.000,A 180.000,B 0.000,C 180.000} C_DIS
LIN {X 113.003,Y 39.300,Z 58.498,A 180.000,B 0.000,C 180.000} C_DIS
; Plunge Move Starts
$VEL.CP=0.01
LIN {X 113.003,Y 39.300,Z 57.625,A 180.000,B 0.000,C 180.000} C_DIS
; Lead In Move Starts
LIN {X 113.003,Y 39.300,Z 56.500,A 180.000,B 0.000,C 180.000} C_DIS
LIN {X 112.866,Y 39.353,Z 56.146,A 180.000,B 0.000,C 180.000} C_DIS
LIN {X 112.537,Y 39.481,Z 56.000,A 180.000,B 0.000,C 180.000} C_DIS
LIN {X 112.203,Y 39.610,Z 56.000,A 180.000,B 0.000,C 180.000} C_DIS
LIN {X 111.820,Y 39.602,Z 56.000,A 180.000,B 0.000,C 180.000} C_DIS
LIN {X 111.556,Y 39.325,Z 56.000,A 180.000,B 0.000,C 180.000} C_DIS
; Cutting Move Starts
$VEL.CP=0.02
LIN {X 111.489,Y 39.154,Z 56.000,A 180.000,B 0.000,C 180.000} C_DIS
LIN {X 111.377,Y 38.841,Z 56.000,A 180.000,B 0.000,C 180.000} C_DIS
LIN {X 111.362,Y 38.796,Z 56.000,A 180.000,B 0.000,C 180.000} C_DIS
LIN {X 111.258,Y 38.439,Z 56.000,A 180.000,B 0.000,C 180.000} C_DIS
LIN {X 111.213,Y 38.260,Z 56.000,A 180.000,B 0.000,C 180.000} C_DIS
LIN {X 111.173,Y 38.081,Z 56.000,A 180.000,B 0.000,C 180.000} C_DIS
LIN {X 111.134,Y 37.902,Z 56.000,A 180.000,B 0.000,C 180.000} C_DIS
LIN {X 111.077,Y 37.545,Z 56.000,A 180.000,B 0.000,C 180.000} C_DIS
LIN {X 111.053,Y 37.366,Z 56.000,A 180.000,B 0.000,C 180.000} C_DIS
LIN {X 111.019,Y 37.006,Z 56.000,A 180.000,B 0.000,C 180.000} C_DIS
LIN {X 111.012,Y 36.830,Z 56.000,A 180.000,B 0.000,C 180.000} C_DIS
LIN {X 111.006,Y 36.651,Z 56.000,A 180.000,B 0.000,C 180.000} C_DIS
LIN {X 111.002,Y 36.472,Z 56.000,A 180.000,B 0.000,C 180.000} C_DIS
LIN {X 111.013,Y 36.115,Z 56.000,A 180.000,B 0.000,C 180.000} C_DIS
LIN {X 111.019,Y 35.994,Z 56.000,A 180.000,B 0.000,C 180.000} C_DIS
LIN {X 111.059,Y 35.578,Z 56.000,A 180.000,B 0.000,C 180.000} C_DIS
LIN {X 111.086,Y 35.400,Z 56.000,A 180.000,B 0.000,C 180.000} C_DIS
LIN {X 111.114,Y 35.221,Z 56.000,A 180.000,B 0.000,C 180.000} C_DIS
LIN {X 111.146,Y 35.042,Z 56.000,A 180.000,B 0.000,C 180.000} C_DIS
LIN {X 111.226,Y 34.685,Z 56.000,A 180.000,B 0.000,C 180.000} C_DIS
LIN {X 111.274,Y 34.506,Z 56.000,A 180.000,B 0.000,C 180.000} C_DIS
LIN {X 111.326,Y 34.327,Z 56.000,A 180.000,B 0.000,C 180.000} C_DIS
LIN {X 111.377,Y 34.159,Z 56.000,A 180.000,B 0.000,C 180.000} C_DIS
LIN {X 111.509,Y 33.791,Z 56.000,A 180.000,B 0.000,C 180.000} C_DIS
LIN {X 111.556,Y 33.675,Z 56.000,A 180.000,B 0.000,C 180.000} C_DIS
LIN {X 111.660,Y 33.433,Z 56.000,A 180.000,B 0.000,C 180.000} C_DIS
LIN {X 111.734,Y 33.269,Z 56.000,A 180.000,B 0.000,C 180.000} C_DIS
LIN {X 111.924,Y 32.897,Z 56.000,A 180.000,B 0.000,C 180.000} C_DIS
LIN {X 112.029,Y 32.718,Z 56.000,A 180.000,B 0.000,C 180.000} C_DIS
LIN {X 112.135,Y 32.539,Z 56.000,A 180.000,B 0.000,C 180.000} C_DIS
LIN {X 112.251,Y 32.361,Z 56.000,A 180.000,B 0.000,C 180.000} C_DIS
LIN {X 112.373,Y 32.182,Z 56.000,A 180.000,B 0.000,C 180.000} C_DIS
LIN {X 112.450,Y 32.072,Z 56.000,A 180.000,B 0.000,C 180.000} C_DIS
LIN {X 112.641,Y 31.824,Z 56.000,A 180.000,B 0.000,C 180.000} C_DIS
LIN {X 112.788,Y 31.646,Z 56.000,A 180.000,B 0.000,C 180.000} C_DIS
LIN {X 112.986,Y 31.421,Z 56.000,A 180.000,B 0.000,C 180.000} C_DIS
LIN {X 113.112,Y 31.288,Z 56.000,A 180.000,B 0.000,C 180.000} C_DIS
LIN {X 113.343,Y 31.057,Z 56.000,A 180.000,B 0.000,C 180.000} C_DIS
LIN {X 113.484,Y 30.930,Z 56.000,A 180.000,B 0.000,C 180.000} C_DIS
LIN {X 113.701,Y 30.739,Z 56.000,A 180.000,B 0.000,C 180.000} C_DIS
LIN {X 113.880,Y 30.598,Z 56.000,A 180.000,B 0.000,C 180.000} C_DIS
LIN {X 114.058,Y 30.460,Z 56.000,A 180.000,B 0.000,C 180.000} C_DIS
LIN {X 114.150,Y 30.394,Z 56.000,A 180.000,B 0.000,C 180.000} C_DIS
LIN {X 114.416,Y 30.213,Z 56.000,A 180.000,B 0.000,C 180.000} C_DIS
LIN {X 114.595,Y 30.102,Z 56.000,A 180.000,B 0.000,C 180.000} C_DIS
LIN {X 114.774,Y 29.996,Z 56.000,A 180.000,B 0.000,C 180.000} C_DIS
LIN {X 114.952,Y 29.896,Z 56.000,A 180.000,B 0.000,C 180.000} C_DIS
LIN {X 115.131,Y 29.805,Z 56.000,A 180.000,B 0.000,C 180.000} C_DIS
LIN {X 115.310,Y 29.714,Z 56.000,A 180.000,B 0.000,C 180.000} C_DIS
LIN {X 115.667,Y 29.559,Z 56.000,A 180.000,B 0.000,C 180.000} C_DIS
LIN {X 115.816,Y 29.500,Z 56.000,A 180.000,B 0.000,C 180.000} C_DIS
LIN {X 116.025,Y 29.425,Z 56.000,A 180.000,B 0.000,C 180.000} C_DIS
LIN {X 116.204,Y 29.362,Z 56.000,A 180.000,B 0.000,C 180.000} C_DIS
LIN {X 116.561,Y 29.258,Z 56.000,A 180.000,B 0.000,C 180.000} C_DIS
LIN {X 116.740,Y 29.213,Z 56.000,A 180.000,B 0.000,C 180.000} C_DIS
LIN {X 117.056,Y 29.143,Z 56.000,A 180.000,B 0.000,C 180.000} C_DIS
LIN {X 117.098,Y 29.134,Z 56.000,A 180.000,B 0.000,C 180.000} C_DIS
LIN {X 117.455,Y 29.077,Z 56.000,A 180.000,B 0.000,C 180.000} C_DIS
LIN {X 117.634,Y 29.053,Z 56.000,A 180.000,B 0.000,C 180.000} C_DIS
LIN {X 117.991,Y 29.020,Z 56.000,A 180.000,B 0.000,C 180.000} C_DIS
LIN {X 118.170,Y 29.012,Z 56.000,A 180.000,B 0.000,C 180.000} C_DIS
LIN {X 118.349,Y 29.006,Z 56.000,A 180.000,B 0.000,C 180.000} C_DIS
LIN {X 118.528,Y 29.002,Z 56.000,A 180.000,B 0.000,C 180.000} C_DIS
LIN {X 118.885,Y 29.013,Z 56.000,A 180.000,B 0.000,C 180.000} C_DIS
LIN {X 119.064,Y 29.025,Z 56.000,A 180.000,B 0.000,C 180.000} C_DIS
LIN {X 119.422,Y 29.059,Z 56.000,A 180.000,B 0.000,C 180.000} C_DIS
LIN {X 119.600,Y 29.086,Z 56.000,A 180.000,B 0.000,C 180.000} C_DIS
LIN {X 119.779,Y 29.114,Z 56.000,A 180.000,B 0.000,C 180.000} C_DIS
LIN {X 119.944,Y 29.143,Z 56.000,A 180.000,B 0.000,C 180.000} C_DIS
LIN {X 120.315,Y 29.226,Z 56.000,A 180.000,B 0.000,C 180.000} C_DIS
LIN {X 120.494,Y 29.274,Z 56.000,A 180.000,B 0.000,C 180.000} C_DIS
LIN {X 120.673,Y 29.326,Z 56.000,A 180.000,B 0.000,C 180.000} C_DIS
LIN {X 120.852,Y 29.381,Z 56.000,A 180.000,B 0.000,C 180.000} C_DIS
LIN {X 121.209,Y 29.509,Z 56.000,A 180.000,B 0.000,C 180.000} C_DIS
LIN {X 121.388,Y 29.583,Z 56.000,A 180.000,B 0.000,C 180.000} C_DIS
LIN {X 121.610,Y 29.679,Z 56.000,A 180.000,B 0.000,C 180.000} C_DIS
LIN {X 121.746,Y 29.742,Z 56.000,A 180.000,B 0.000,C 180.000} C_DIS
LIN {X 122.103,Y 29.924,Z 56.000,A 180.000,B 0.000,C 180.000} C_DIS
LIN {X 122.282,Y 30.029,Z 56.000,A 180.000,B 0.000,C 180.000} C_DIS
LIN {X 122.461,Y 30.135,Z 56.000,A 180.000,B 0.000,C 180.000} C_DIS
LIN {X 122.587,Y 30.215,Z 56.000,A 180.000,B 0.000,C 180.000} C_DIS
LIN {X 122.850,Y 30.394,Z 56.000,A 180.000,B 0.000,C 180.000} C_DIS
LIN {X 122.997,Y 30.503,Z 56.000,A 180.000,B 0.000,C 180.000} C_DIS
LIN {X 123.176,Y 30.641,Z 56.000,A 180.000,B 0.000,C 180.000} C_DIS
LIN {X 123.313,Y 30.752,Z 56.000,A 180.000,B 0.000,C 180.000} C_DIS
LIN {X 123.533,Y 30.945,Z 56.000,A 180.000,B 0.000,C 180.000} C_DIS
LIN {X 123.709,Y 31.109,Z 56.000,A 180.000,B 0.000,C 180.000} C_DIS
LIN {X 123.891,Y 31.291,Z 56.000,A 180.000,B 0.000,C 180.000} C_DIS
LIN {X 124.055,Y 31.467,Z 56.000,A 180.000,B 0.000,C 180.000} C_DIS
LIN {X 124.248,Y 31.687,Z 56.000,A 180.000,B 0.000,C 180.000} C_DIS
LIN {X 124.359,Y 31.824,Z 56.000,A 180.000,B 0.000,C 180.000} C_DIS
LIN {X 124.497,Y 32.003,Z 56.000,A 180.000,B 0.000,C 180.000} C_DIS
LIN {X 124.606,Y 32.150,Z 56.000,A 180.000,B 0.000,C 180.000} C_DIS
LIN {X 124.785,Y 32.413,Z 56.000,A 180.000,B 0.000,C 180.000} C_DIS
LIN {X 124.865,Y 32.539,Z 56.000,A 180.000,B 0.000,C 180.000} C_DIS
LIN {X 124.971,Y 32.718,Z 56.000,A 180.000,B 0.000,C 180.000} C_DIS
LIN {X 125.076,Y 32.897,Z 56.000,A 180.000,B 0.000,C 180.000} C_DIS
LIN {X 125.258,Y 33.254,Z 56.000,A 180.000,B 0.000,C 180.000} C_DIS
LIN {X 125.321,Y 33.390,Z 56.000,A 180.000,B 0.000,C 180.000} C_DIS
LIN {X 125.417,Y 33.612,Z 56.000,A 180.000,B 0.000,C 180.000} C_DIS
LIN {X 125.491,Y 33.791,Z 56.000,A 180.000,B 0.000,C 180.000} C_DIS
LIN {X 125.619,Y 34.148,Z 56.000,A 180.000,B 0.000,C 180.000} C_DIS
LIN {X 125.674,Y 34.327,Z 56.000,A 180.000,B 0.000,C 180.000} C_DIS
LIN {X 125.726,Y 34.506,Z 56.000,A 180.000,B 0.000,C 180.000} C_DIS
LIN {X 125.774,Y 34.685,Z 56.000,A 180.000,B 0.000,C 180.000} C_DIS
LIN {X 125.857,Y 35.056,Z 56.000,A 180.000,B 0.000,C 180.000} C_DIS
LIN {X 125.886,Y 35.221,Z 56.000,A 180.000,B 0.000,C 180.000} C_DIS
LIN {X 125.914,Y 35.400,Z 56.000,A 180.000,B 0.000,C 180.000} C_DIS
LIN {X 125.941,Y 35.578,Z 56.000,A 180.000,B 0.000,C 180.000} C_DIS
LIN {X 125.975,Y 35.936,Z 56.000,A 180.000,B 0.000,C 180.000} C_DIS
LIN {X 125.987,Y 36.115,Z 56.000,A 180.000,B 0.000,C 180.000} C_DIS
LIN {X 125.998,Y 36.472,Z 56.000,A 180.000,B 0.000,C 180.000} C_DIS
LIN {X 125.994,Y 36.651,Z 56.000,A 180.000,B 0.000,C 180.000} C_DIS
LIN {X 125.988,Y 36.830,Z 56.000,A 180.000,B 0.000,C 180.000} C_DIS
LIN {X 125.980,Y 37.009,Z 56.000,A 180.000,B 0.000,C 180.000} C_DIS
LIN {X 125.947,Y 37.366,Z 56.000,A 180.000,B 0.000,C 180.000} C_DIS
LIN {X 125.923,Y 37.545,Z 56.000,A 180.000,B 0.000,C 180.000} C_DIS
LIN {X 125.866,Y 37.902,Z 56.000,A 180.000,B 0.000,C 180.000} C_DIS
LIN {X 125.857,Y 37.944,Z 56.000,A 180.000,B 0.000,C 180.000} C_DIS
LIN {X 125.787,Y 38.260,Z 56.000,A 180.000,B 0.000,C 180.000} C_DIS
LIN {X 125.742,Y 38.439,Z 56.000,A 180.000,B 0.000,C 180.000} C_DIS
LIN {X 125.638,Y 38.796,Z 56.000,A 180.000,B 0.000,C 180.000} C_DIS
LIN {X 125.575,Y 38.975,Z 56.000,A 180.000,B 0.000,C 180.000} C_DIS
LIN {X 125.500,Y 39.184,Z 56.000,A 180.000,B 0.000,C 180.000} C_DIS
LIN {X 125.441,Y 39.333,Z 56.000,A 180.000,B 0.000,C 180.000} C_DIS
LIN {X 125.286,Y 39.690,Z 56.000,A 180.000,B 0.000,C 180.000} C_DIS
LIN {X 125.195,Y 39.869,Z 56.000,A 180.000,B 0.000,C 180.000} C_DIS
LIN {X 125.104,Y 40.048,Z 56.000,A 180.000,B 0.000,C 180.000} C_DIS
LIN {X 125.004,Y 40.226,Z 56.000,A 180.000,B 0.000,C 180.000} C_DIS
LIN {X 124.898,Y 40.405,Z 56.000,A 180.000,B 0.000,C 180.000} C_DIS
LIN {X 124.787,Y 40.584,Z 56.000,A 180.000,B 0.000,C 180.000} C_DIS
LIN {X 124.606,Y 40.850,Z 56.000,A 180.000,B 0.000,C 180.000} C_DIS
LIN {X 124.540,Y 40.942,Z 56.000,A 180.000,B 0.000,C 180.000} C_DIS
LIN {X 124.402,Y 41.120,Z 56.000,A 180.000,B 0.000,C 180.000} C_DIS
LIN {X 124.261,Y 41.299,Z 56.000,A 180.000,B 0.000,C 180.000} C_DIS
LIN {X 124.070,Y 41.516,Z 56.000,A 180.000,B 0.000,C 180.000} C_DIS
LIN {X 123.943,Y 41.657,Z 56.000,A 180.000,B 0.000,C 180.000} C_DIS
LIN {X 123.712,Y 41.888,Z 56.000,A 180.000,B 0.000,C 180.000} C_DIS
LIN {X 123.579,Y 42.014,Z 56.000,A 180.000,B 0.000,C 180.000} C_DIS
LIN {X 123.354,Y 42.212,Z 56.000,A 180.000,B 0.000,C 180.000} C_DIS
LIN {X 123.176,Y 42.359,Z 56.000,A 180.000,B 0.000,C 180.000} C_DIS
LIN {X 122.928,Y 42.550,Z 56.000,A 180.000,B 0.000,C 180.000} C_DIS
LIN {X 122.818,Y 42.627,Z 56.000,A 180.000,B 0.000,C 180.000} C_DIS
LIN {X 122.639,Y 42.749,Z 56.000,A 180.000,B 0.000,C 180.000} C_DIS
LIN {X 122.461,Y 42.865,Z 56.000,A 180.000,B 0.000,C 180.000} C_DIS
LIN {X 122.282,Y 42.971,Z 56.000,A 180.000,B 0.000,C 180.000} C_DIS
LIN {X 122.103,Y 43.076,Z 56.000,A 180.000,B 0.000,C 180.000} C_DIS
LIN {X 121.731,Y 43.266,Z 56.000,A 180.000,B 0.000,C 180.000} C_DIS
LIN {X 121.567,Y 43.340,Z 56.000,A 180.000,B 0.000,C 180.000} C_DIS
LIN {X 121.325,Y 43.444,Z 56.000,A 180.000,B 0.000,C 180.000} C_DIS
LIN {X 121.209,Y 43.491,Z 56.000,A 180.000,B 0.000,C 180.000} C_DIS
LIN {X 120.841,Y 43.623,Z 56.000,A 180.000,B 0.000,C 180.000} C_DIS
LIN {X 120.673,Y 43.674,Z 56.000,A 180.000,B 0.000,C 180.000} C_DIS
LIN {X 120.494,Y 43.726,Z 56.000,A 180.000,B 0.000,C 180.000} C_DIS
LIN {X 120.315,Y 43.774,Z 56.000,A 180.000,B 0.000,C 180.000} C_DIS
LIN {X 119.958,Y 43.854,Z 56.000,A 180.000,B 0.000,C 180.000} C_DIS
LIN {X 119.779,Y 43.886,Z 56.000,A 180.000,B 0.000,C 180.000} C_DIS
LIN {X 119.600,Y 43.914,Z 56.000,A 180.000,B 0.000,C 180.000} C_DIS
LIN {X 119.422,Y 43.941,Z 56.000,A 180.000,B 0.000,C 180.000} C_DIS
LIN {X 119.006,Y 43.981,Z 56.000,A 180.000,B 0.000,C 180.000} C_DIS
LIN {X 118.885,Y 43.987,Z 56.000,A 180.000,B 0.000,C 180.000} C_DIS
LIN {X 118.528,Y 43.998,Z 56.000,A 180.000,B 0.000,C 180.000} C_DIS
LIN {X 118.349,Y 43.994,Z 56.000,A 180.000,B 0.000,C 180.000} C_DIS
LIN {X 118.170,Y 43.988,Z 56.000,A 180.000,B 0.000,C 180.000} C_DIS
LIN {X 117.994,Y 43.981,Z 56.000,A 180.000,B 0.000,C 180.000} C_DIS
LIN {X 117.634,Y 43.947,Z 56.000,A 180.000,B 0.000,C 180.000} C_DIS
LIN {X 117.455,Y 43.923,Z 56.000,A 180.000,B 0.000,C 180.000} C_DIS
LIN {X 117.098,Y 43.866,Z 56.000,A 180.000,B 0.000,C 180.000} C_DIS
LIN {X 116.919,Y 43.827,Z 56.000,A 180.000,B 0.000,C 180.000} C_DIS
LIN {X 116.740,Y 43.787,Z 56.000,A 180.000,B 0.000,C 180.000} C_DIS
LIN {X 116.561,Y 43.742,Z 56.000,A 180.000,B 0.000,C 180.000} C_DIS
LIN {X 116.204,Y 43.638,Z 56.000,A 180.000,B 0.000,C 180.000} C_DIS
LIN {X 116.159,Y 43.623,Z 56.000,A 180.000,B 0.000,C 180.000} C_DIS
LIN {X 115.846,Y 43.511,Z 56.000,A 180.000,B 0.000,C 180.000} C_DIS
LIN {X 115.675,Y 43.444,Z 56.000,A 180.000,B 0.000,C 180.000} C_DIS
LIN {X 115.310,Y 43.286,Z 56.000,A 180.000,B 0.000,C 180.000} C_DIS
LIN {X 115.269,Y 43.266,Z 56.000,A 180.000,B 0.000,C 180.000} C_DIS
LIN {X 114.918,Y 43.087,Z 56.000,A 180.000,B 0.000,C 180.000} C_DIS
LIN {X 114.774,Y 43.004,Z 56.000,A 180.000,B 0.000,C 180.000} C_DIS
LIN {X 114.595,Y 42.898,Z 56.000,A 180.000,B 0.000,C 180.000} C_DIS
LIN {X 114.416,Y 42.787,Z 56.000,A 180.000,B 0.000,C 180.000} C_DIS
LIN {X 114.237,Y 42.665,Z 56.000,A 180.000,B 0.000,C 180.000} C_DIS
LIN {X 114.072,Y 42.550,Z 56.000,A 180.000,B 0.000,C 180.000} C_DIS
LIN {X 113.841,Y 42.372,Z 56.000,A 180.000,B 0.000,C 180.000} C_DIS
LIN {X 113.701,Y 42.261,Z 56.000,A 180.000,B 0.000,C 180.000} C_DIS
LIN {X 113.421,Y 42.014,Z 56.000,A 180.000,B 0.000,C 180.000} C_DIS
LIN {X 113.343,Y 41.943,Z 56.000,A 180.000,B 0.000,C 180.000} C_DIS
LIN {X 113.057,Y 41.657,Z 56.000,A 180.000,B 0.000,C 180.000} C_DIS
LIN {X 112.986,Y 41.579,Z 56.000,A 180.000,B 0.000,C 180.000} C_DIS
LIN {X 112.739,Y 41.299,Z 56.000,A 180.000,B 0.000,C 180.000} C_DIS
LIN {X 112.628,Y 41.159,Z 56.000,A 180.000,B 0.000,C 180.000} C_DIS
LIN {X 112.450,Y 40.928,Z 56.000,A 180.000,B 0.000,C 180.000} C_DIS
LIN {X 112.335,Y 40.763,Z 56.000,A 180.000,B 0.000,C 180.000} C_DIS
LIN {X 112.213,Y 40.584,Z 56.000,A 180.000,B 0.000,C 180.000} C_DIS
LIN {X 112.102,Y 40.405,Z 56.000,A 180.000,B 0.000,C 180.000} C_DIS
LIN {X 111.996,Y 40.226,Z 56.000,A 180.000,B 0.000,C 180.000} C_DIS
LIN {X 111.913,Y 40.082,Z 56.000,A 180.000,B 0.000,C 180.000} C_DIS
LIN {X 111.734,Y 39.731,Z 56.000,A 180.000,B 0.000,C 180.000} C_DIS
LIN {X 111.714,Y 39.690,Z 56.000,A 180.000,B 0.000,C 180.000} C_DIS
LIN {X 111.556,Y 39.325,Z 56.000,A 180.000,B 0.000,C 180.000} C_DIS
; Link Move Starts
LIN {X 111.445,Y 39.030,Z 56.000,A 180.000,B 0.000,C 180.000} C_DIS
LIN {X 111.343,Y 38.732,Z 55.999,A 180.000,B 0.000,C 180.000} C_DIS
LIN {X 111.256,Y 38.429,Z 55.998,A 180.000,B 0.000,C 180.000} C_DIS
LIN {X 111.183,Y 38.123,Z 55.996,A 180.000,B 0.000,C 180.000} C_DIS
LIN {X 111.120,Y 37.814,Z 55.994,A 180.000,B 0.000,C 180.000} C_DIS
LIN {X 111.070,Y 37.503,Z 55.991,A 180.000,B 0.000,C 180.000} C_DIS
LIN {X 111.037,Y 37.190,Z 55.988,A 180.000,B 0.000,C 180.000} C_DIS
LIN {X 111.013,Y 36.876,Z 55.985,A 180.000,B 0.000,C 180.000} C_DIS
LIN {X 111.003,Y 36.561,Z 55.981,A 180.000,B 0.000,C 180.000} C_DIS
LIN {X 111.009,Y 36.246,Z 55.977,A 180.000,B 0.000,C 180.000} C_DIS
LIN {X 111.025,Y 35.932,Z 55.972,A 180.000,B 0.000,C 180.000} C_DIS
LIN {X 111.040,Y 35.775,Z 55.969,A 180.000,B 0.000,C 180.000} C_DIS
LIN {X 111.055,Y 35.618,Z 55.967,A 180.000,B 0.000,C 180.000} C_DIS
LIN {X 111.076,Y 35.462,Z 55.964,A 180.000,B 0.000,C 180.000} C_DIS
LIN {X 111.101,Y 35.307,Z 55.961,A 180.000,B 0.000,C 180.000} C_DIS
LIN {X 111.125,Y 35.151,Z 55.959,A 180.000,B 0.000,C 180.000} C_DIS
LIN {X 111.156,Y 34.997,Z 55.956,A 180.000,B 0.000,C 180.000} C_DIS
LIN {X 111.190,Y 34.843,Z 55.952,A 180.000,B 0.000,C 180.000} C_DIS
LIN {X 111.225,Y 34.689,Z 55.949,A 180.000,B 0.000,C 180.000} C_DIS
LIN {X 111.265,Y 34.537,Z 55.946,A 180.000,B 0.000,C 180.000} C_DIS
LIN {X 111.309,Y 34.386,Z 55.943,A 180.000,B 0.000,C 180.000} C_DIS
LIN {X 111.353,Y 34.235,Z 55.939,A 180.000,B 0.000,C 180.000} C_DIS
LIN {X 111.403,Y 34.085,Z 55.936,A 180.000,B 0.000,C 180.000} C_DIS
LIN {X 111.457,Y 33.937,Z 55.932,A 180.000,B 0.000,C 180.000} C_DIS
LIN {X 111.510,Y 33.789,Z 55.928,A 180.000,B 0.000,C 180.000} C_DIS
LIN {X 111.570,Y 33.643,Z 55.925,A 180.000,B 0.000,C 180.000} C_DIS
LIN {X 111.632,Y 33.499,Z 55.921,A 180.000,B 0.000,C 180.000} C_DIS
LIN {X 111.695,Y 33.354,Z 55.917,A 180.000,B 0.000,C 180.000} C_DIS
LIN {X 111.763,Y 33.212,Z 55.913,A 180.000,B 0.000,C 180.000} C_DIS
LIN {X 111.835,Y 33.072,Z 55.909,A 180.000,B 0.000,C 180.000} C_DIS
LIN {X 111.906,Y 32.932,Z 55.905,A 180.000,B 0.000,C 180.000} C_DIS
LIN {X 111.984,Y 32.794,Z 55.900,A 180.000,B 0.000,C 180.000} C_DIS
LIN {X 112.064,Y 32.659,Z 55.896,A 180.000,B 0.000,C 180.000} C_DIS
LIN {X 112.144,Y 32.523,Z 55.892,A 180.000,B 0.000,C 180.000} C_DIS
LIN {X 112.230,Y 32.391,Z 55.887,A 180.000,B 0.000,C 180.000} C_DIS
LIN {X 112.319,Y 32.261,Z 55.883,A 180.000,B 0.000,C 180.000} C_DIS
LIN {X 112.407,Y 32.131,Z 55.878,A 180.000,B 0.000,C 180.000} C_DIS
LIN {X 112.501,Y 32.005,Z 55.873,A 180.000,B 0.000,C 180.000} C_DIS
LIN {X 112.598,Y 31.880,Z 55.869,A 180.000,B 0.000,C 180.000} C_DIS
LIN {X 112.694,Y 31.756,Z 55.864,A 180.000,B 0.000,C 180.000} C_DIS
LIN {X 112.796,Y 31.636,Z 55.859,A 180.000,B 0.000,C 180.000} C_DIS
LIN {X 112.901,Y 31.518,Z 55.854,A 180.000,B 0.000,C 180.000} C_DIS
LIN {X 112.953,Y 31.459,Z 55.851,A 180.000,B 0.000,C 180.000} C_DIS
LIN {X 113.005,Y 31.399,Z 55.849,A 180.000,B 0.000,C 180.000} C_DIS
LIN {X 113.059,Y 31.342,Z 55.846,A 180.000,B 0.000,C 180.000} C_DIS
LIN {X 113.114,Y 31.286,Z 55.844,A 180.000,B 0.000,C 180.000} C_DIS
LIN {X 113.170,Y 31.230,Z 55.841,A 180.000,B 0.000,C 180.000} C_DIS
LIN {X 113.226,Y 31.175,Z 55.839,A 180.000,B 0.000,C 180.000} C_DIS
LIN {X 113.281,Y 31.119,Z 55.836,A 180.000,B 0.000,C 180.000} C_DIS
LIN {X 113.337,Y 31.063,Z 55.833,A 180.000,B 0.000,C 180.000} C_DIS
LIN {X 113.394,Y 31.009,Z 55.831,A 180.000,B 0.000,C 180.000} C_DIS
LIN {X 113.512,Y 30.905,Z 55.825,A 180.000,B 0.000,C 180.000} C_DIS
LIN {X 113.631,Y 30.801,Z 55.820,A 180.000,B 0.000,C 180.000} C_DIS
LIN {X 113.690,Y 30.749,Z 55.817,A 180.000,B 0.000,C 180.000} C_DIS
LIN {X 113.750,Y 30.699,Z 55.815,A 180.000,B 0.000,C 180.000} C_DIS
LIN {X 113.875,Y 30.602,Z 55.809,A 180.000,B 0.000,C 180.000} C_DIS
LIN {X 113.937,Y 30.554,Z 55.806,A 180.000,B 0.000,C 180.000} C_DIS
LIN {X 114.061,Y 30.457,Z 55.801,A 180.000,B 0.000,C 180.000} C_DIS
LIN {X 114.125,Y 30.411,Z 55.798,A 180.000,B 0.000,C 180.000} C_DIS
LIN {X 114.190,Y 30.367,Z 55.796,A 180.000,B 0.000,C 180.000} C_DIS
LIN {X 114.321,Y 30.278,Z 55.790,A 180.000,B 0.000,C 180.000} C_DIS
LIN {X 114.451,Y 30.190,Z 55.785,A 180.000,B 0.000,C 180.000} C_DIS
LIN {X 114.517,Y 30.148,Z 55.782,A 180.000,B 0.000,C 180.000} C_DIS
LIN {X 114.653,Y 30.067,Z 55.776,A 180.000,B 0.000,C 180.000} C_DIS
LIN {X 114.721,Y 30.027,Z 55.774,A 180.000,B 0.000,C 180.000} C_DIS
LIN {X 114.856,Y 29.947,Z 55.768,A 180.000,B 0.000,C 180.000} C_DIS
LIN {X 114.925,Y 29.909,Z 55.765,A 180.000,B 0.000,C 180.000} C_DIS
LIN {X 114.996,Y 29.874,Z 55.763,A 180.000,B 0.000,C 180.000} C_DIS
LIN {X 115.136,Y 29.802,Z 55.757,A 180.000,B 0.000,C 180.000} C_DIS
LIN {X 115.276,Y 29.731,Z 55.752,A 180.000,B 0.000,C 180.000} C_DIS
LIN {X 115.348,Y 29.697,Z 55.749,A 180.000,B 0.000,C 180.000} C_DIS
LIN {X 115.492,Y 29.635,Z 55.743,A 180.000,B 0.000,C 180.000} C_DIS
LIN {X 115.564,Y 29.604,Z 55.741,A 180.000,B 0.000,C 180.000} C_DIS
LIN {X 115.709,Y 29.541,Z 55.735,A 180.000,B 0.000,C 180.000} C_DIS
LIN {X 115.782,Y 29.512,Z 55.732,A 180.000,B 0.000,C 180.000} C_DIS
LIN {X 115.856,Y 29.486,Z 55.730,A 180.000,B 0.000,C 180.000} C_DIS
LIN {X 116.005,Y 29.432,Z 55.724,A 180.000,B 0.000,C 180.000} C_DIS
LIN {X 116.153,Y 29.379,Z 55.719,A 180.000,B 0.000,C 180.000} C_DIS
LIN {X 116.228,Y 29.355,Z 55.716,A 180.000,B 0.000,C 180.000} C_DIS
LIN {X 116.379,Y 29.311,Z 55.710,A 180.000,B 0.000,C 180.000} C_DIS
LIN {X 116.455,Y 29.289,Z 55.708,A 180.000,B 0.000,C 180.000} C_DIS
LIN {X 116.606,Y 29.245,Z 55.702,A 180.000,B 0.000,C 180.000} C_DIS
LIN {X 116.682,Y 29.226,Z 55.699,A 180.000,B 0.000,C 180.000} C_DIS
LIN {X 116.759,Y 29.209,Z 55.697,A 180.000,B 0.000,C 180.000} C_DIS
LIN {X 116.913,Y 29.175,Z 55.691,A 180.000,B 0.000,C 180.000} C_DIS
LIN {X 117.067,Y 29.140,Z 55.686,A 180.000,B 0.000,C 180.000} C_DIS
LIN {X 117.144,Y 29.126,Z 55.683,A 180.000,B 0.000,C 180.000} C_DIS
LIN {X 117.300,Y 29.102,Z 55.677,A 180.000,B 0.000,C 180.000} C_DIS
LIN {X 117.378,Y 29.089,Z 55.675,A 180.000,B 0.000,C 180.000} C_DIS
LIN {X 117.533,Y 29.065,Z 55.669,A 180.000,B 0.000,C 180.000} C_DIS
LIN {X 117.611,Y 29.056,Z 55.666,A 180.000,B 0.000,C 180.000} C_DIS
LIN {X 117.768,Y 29.041,Z 55.661,A 180.000,B 0.000,C 180.000} C_DIS
LIN {X 118.003,Y 29.018,Z 55.653,A 180.000,B 0.000,C 180.000} C_DIS
LIN {X 118.082,Y 29.014,Z 55.650,A 180.000,B 0.000,C 180.000} C_DIS
LIN {X 118.476,Y 29.002,Z 55.636,A 180.000,B 0.000,C 180.000} C_DIS
LIN {X 118.554,Y 29.003,Z 55.633,A 180.000,B 0.000,C 180.000} C_DIS
LIN {X 118.712,Y 29.008,Z 55.628,A 180.000,B 0.000,C 180.000} C_DIS
LIN {X 118.948,Y 29.015,Z 55.620,A 180.000,B 0.000,C 180.000} C_DIS
LIN {X 119.026,Y 29.021,Z 55.617,A 180.000,B 0.000,C 180.000} C_DIS
LIN {X 119.418,Y 29.058,Z 55.603,A 180.000,B 0.000,C 180.000} C_DIS
LIN {X 119.496,Y 29.069,Z 55.600,A 180.000,B 0.000,C 180.000} C_DIS
LIN {X 119.885,Y 29.131,Z 55.587,A 180.000,B 0.000,C 180.000} C_DIS
LIN {X 119.962,Y 29.147,Z 55.584,A 180.000,B 0.000,C 180.000} C_DIS
LIN {X 120.347,Y 29.233,Z 55.570,A 180.000,B 0.000,C 180.000} C_DIS
LIN {X 120.423,Y 29.254,Z 55.567,A 180.000,B 0.000,C 180.000} C_DIS
LIN {X 120.801,Y 29.363,Z 55.554,A 180.000,B 0.000,C 180.000} C_DIS
LIN {X 120.875,Y 29.389,Z 55.551,A 180.000,B 0.000,C 180.000} C_DIS
LIN {X 121.246,Y 29.523,Z 55.537,A 180.000,B 0.000,C 180.000} C_DIS
LIN {X 121.318,Y 29.553,Z 55.534,A 180.000,B 0.000,C 180.000} C_DIS
LIN {X 121.680,Y 29.709,Z 55.521,A 180.000,B 0.000,C 180.000} C_DIS
LIN {X 121.750,Y 29.744,Z 55.518,A 180.000,B 0.000,C 180.000} C_DIS
LIN {X 122.101,Y 29.923,Z 55.504,A 180.000,B 0.000,C 180.000} C_DIS
LIN {X 122.169,Y 29.962,Z 55.501,A 180.000,B 0.000,C 180.000} C_DIS
LIN {X 122.508,Y 30.163,Z 55.488,A 180.000,B 0.000,C 180.000} C_DIS
LIN {X 122.574,Y 30.207,Z 55.485,A 180.000,B 0.000,C 180.000} C_DIS
LIN {X 122.900,Y 30.428,Z 55.471,A 180.000,B 0.000,C 180.000} C_DIS
LIN {X 122.962,Y 30.476,Z 55.468,A 180.000,B 0.000,C 180.000} C_DIS
LIN {X 123.273,Y 30.717,Z 55.455,A 180.000,B 0.000,C 180.000} C_DIS
LIN {X 123.333,Y 30.769,Z 55.452,A 180.000,B 0.000,C 180.000} C_DIS
LIN {X 123.628,Y 31.029,Z 55.438,A 180.000,B 0.000,C 180.000} C_DIS
LIN {X 123.684,Y 31.085,Z 55.435,A 180.000,B 0.000,C 180.000} C_DIS
LIN {X 123.907,Y 31.307,Z 55.424,A 180.000,B 0.000,C 180.000} C_DIS
LIN {X 123.963,Y 31.363,Z 55.422,A 180.000,B 0.000,C 180.000} C_DIS
LIN {X 124.015,Y 31.422,Z 55.419,A 180.000,B 0.000,C 180.000} C_DIS
LIN {X 124.275,Y 31.717,Z 55.405,A 180.000,B 0.000,C 180.000} C_DIS
LIN {X 124.324,Y 31.779,Z 55.402,A 180.000,B 0.000,C 180.000} C_DIS
LIN {X 124.421,Y 31.904,Z 55.397,A 180.000,B 0.000,C 180.000} C_DIS
LIN {X 124.565,Y 32.091,Z 55.389,A 180.000,B 0.000,C 180.000} C_DIS
LIN {X 124.610,Y 32.156,Z 55.386,A 180.000,B 0.000,C 180.000} C_DIS
LIN {X 124.831,Y 32.481,Z 55.372,A 180.000,B 0.000,C 180.000} C_DIS
LIN {X 124.871,Y 32.549,Z 55.369,A 180.000,B 0.000,C 180.000} C_DIS
LIN {X 124.951,Y 32.685,Z 55.364,A 180.000,B 0.000,C 180.000} C_DIS
LIN {X 125.032,Y 32.820,Z 55.358,A 180.000,B 0.000,C 180.000} C_DIS
LIN {X 125.072,Y 32.888,Z 55.356,A 180.000,B 0.000,C 180.000} C_DIS
LIN {X 125.179,Y 33.099,Z 55.347,A 180.000,B 0.000,C 180.000} C_DIS
LIN {X 125.250,Y 33.239,Z 55.342,A 180.000,B 0.000,C 180.000} C_DIS
LIN {X 125.286,Y 33.309,Z 55.339,A 180.000,B 0.000,C 180.000} C_DIS
LIN {X 125.442,Y 33.671,Z 55.325,A 180.000,B 0.000,C 180.000} C_DIS
LIN {X 125.473,Y 33.743,Z 55.323,A 180.000,B 0.000,C 180.000} C_DIS
LIN {X 125.527,Y 33.891,Z 55.317,A 180.000,B 0.000,C 180.000} C_DIS
LIN {X 125.607,Y 34.114,Z 55.309,A 180.000,B 0.000,C 180.000} C_DIS
LIN {X 125.633,Y 34.188,Z 55.306,A 180.000,B 0.000,C 180.000} C_DIS
LIN {X 125.699,Y 34.415,Z 55.298,A 180.000,B 0.000,C 180.000} C_DIS
LIN {X 125.743,Y 34.566,Z 55.292,A 180.000,B 0.000,C 180.000} C_DIS
LIN {X 125.765,Y 34.642,Z 55.290,A 180.000,B 0.000,C 180.000} C_DIS
LIN {X 125.799,Y 34.795,Z 55.284,A 180.000,B 0.000,C 180.000} C_DIS
LIN {X 125.851,Y 35.026,Z 55.276,A 180.000,B 0.000,C 180.000} C_DIS
LIN {X 125.867,Y 35.103,Z 55.273,A 180.000,B 0.000,C 180.000} C_DIS
LIN {X 125.904,Y 35.336,Z 55.265,A 180.000,B 0.000,C 180.000} C_DIS
LIN {X 125.929,Y 35.492,Z 55.259,A 180.000,B 0.000,C 180.000} C_DIS
LIN {X 125.941,Y 35.570,Z 55.257,A 180.000,B 0.000,C 180.000} C_DIS
LIN {X 125.955,Y 35.727,Z 55.251,A 180.000,B 0.000,C 180.000} C_DIS
LIN {X 125.978,Y 35.962,Z 55.243,A 180.000,B 0.000,C 180.000} C_DIS
LIN {X 125.984,Y 36.040,Z 55.240,A 180.000,B 0.000,C 180.000} C_DIS
LIN {X 125.992,Y 36.276,Z 55.232,A 180.000,B 0.000,C 180.000} C_DIS
LIN {X 125.997,Y 36.434,Z 55.226,A 180.000,B 0.000,C 180.000} C_DIS
LIN {X 125.998,Y 36.513,Z 55.224,A 180.000,B 0.000,C 180.000} C_DIS
LIN {X 125.993,Y 36.670,Z 55.218,A 180.000,B 0.000,C 180.000} C_DIS
LIN {X 125.986,Y 36.906,Z 55.210,A 180.000,B 0.000,C 180.000} C_DIS
LIN {X 125.983,Y 36.985,Z 55.207,A 180.000,B 0.000,C 180.000} C_DIS
LIN {X 125.960,Y 37.220,Z 55.199,A 180.000,B 0.000,C 180.000} C_DIS
LIN {X 125.946,Y 37.377,Z 55.193,A 180.000,B 0.000,C 180.000} C_DIS
LIN {X 125.937,Y 37.455,Z 55.191,A 180.000,B 0.000,C 180.000} C_DIS
LIN {X 125.913,Y 37.611,Z 55.185,A 180.000,B 0.000,C 180.000} C_DIS
LIN {X 125.888,Y 37.766,Z 55.180,A 180.000,B 0.000,C 180.000} C_DIS
LIN {X 125.876,Y 37.844,Z 55.177,A 180.000,B 0.000,C 180.000} C_DIS
LIN {X 125.862,Y 37.922,Z 55.174,A 180.000,B 0.000,C 180.000} C_DIS
LIN {X 125.828,Y 38.075,Z 55.169,A 180.000,B 0.000,C 180.000} C_DIS
LIN {X 125.794,Y 38.229,Z 55.164,A 180.000,B 0.000,C 180.000} C_DIS
LIN {X 125.776,Y 38.306,Z 55.161,A 180.000,B 0.000,C 180.000} C_DIS
LIN {X 125.758,Y 38.383,Z 55.159,A 180.000,B 0.000,C 180.000} C_DIS
LIN {X 125.736,Y 38.458,Z 55.156,A 180.000,B 0.000,C 180.000} C_DIS
LIN {X 125.714,Y 38.534,Z 55.154,A 180.000,B 0.000,C 180.000} C_DIS
LIN {X 125.692,Y 38.610,Z 55.151,A 180.000,B 0.000,C 180.000} C_DIS
LIN {X 125.670,Y 38.685,Z 55.149,A 180.000,B 0.000,C 180.000} C_DIS
LIN {X 125.625,Y 38.836,Z 55.144,A 180.000,B 0.000,C 180.000} C_DIS
LIN {X 125.572,Y 38.984,Z 55.139,A 180.000,B 0.000,C 180.000} C_DIS
LIN {X 125.518,Y 39.132,Z 55.134,A 180.000,B 0.000,C 180.000} C_DIS
LIN {X 125.464,Y 39.280,Z 55.129,A 180.000,B 0.000,C 180.000} C_DIS
LIN {X 125.401,Y 39.425,Z 55.124,A 180.000,B 0.000,C 180.000} C_DIS
LIN {X 125.339,Y 39.569,Z 55.120,A 180.000,B 0.000,C 180.000} C_DIS
LIN {X 125.275,Y 39.713,Z 55.115,A 180.000,B 0.000,C 180.000} C_DIS
LIN {X 125.203,Y 39.854,Z 55.111,A 180.000,B 0.000,C 180.000} C_DIS
LIN {X 125.132,Y 39.994,Z 55.106,A 180.000,B 0.000,C 180.000} C_DIS
LIN {X 125.059,Y 40.134,Z 55.102,A 180.000,B 0.000,C 180.000} C_DIS
LIN {X 124.979,Y 40.269,Z 55.097,A 180.000,B 0.000,C 180.000} C_DIS
LIN {X 124.898,Y 40.405,Z 55.093,A 180.000,B 0.000,C 180.000} C_DIS
LIN {X 124.817,Y 40.539,Z 55.089,A 180.000,B 0.000,C 180.000} C_DIS
LIN {X 124.728,Y 40.670,Z 55.085,A 180.000,B 0.000,C 180.000} C_DIS
LIN {X 124.640,Y 40.800,Z 55.081,A 180.000,B 0.000,C 180.000} C_DIS
LIN {X 124.550,Y 40.929,Z 55.077,A 180.000,B 0.000,C 180.000} C_DIS
LIN {X 124.453,Y 41.054,Z 55.073,A 180.000,B 0.000,C 180.000} C_DIS
LIN {X 124.357,Y 41.178,Z 55.070,A 180.000,B 0.000,C 180.000} C_DIS
LIN {X 124.259,Y 41.302,Z 55.066,A 180.000,B 0.000,C 180.000} C_DIS
LIN {X 124.155,Y 41.420,Z 55.062,A 180.000,B 0.000,C 180.000} C_DIS
LIN {X 124.051,Y 41.538,Z 55.059,A 180.000,B 0.000,C 180.000} C_DIS
LIN {X 123.945,Y 41.655,Z 55.056,A 180.000,B 0.000,C 180.000} C_DIS
LIN {X 123.834,Y 41.766,Z 55.052,A 180.000,B 0.000,C 180.000} C_DIS
LIN {X 123.722,Y 41.877,Z 55.049,A 180.000,B 0.000,C 180.000} C_DIS
LIN {X 123.609,Y 41.987,Z 55.046,A 180.000,B 0.000,C 180.000} C_DIS
LIN {X 123.491,Y 42.092,Z 55.043,A 180.000,B 0.000,C 180.000} C_DIS
LIN {X 123.373,Y 42.196,Z 55.040,A 180.000,B 0.000,C 180.000} C_DIS
LIN {X 123.254,Y 42.298,Z 55.037,A 180.000,B 0.000,C 180.000} C_DIS
LIN {X 123.129,Y 42.395,Z 55.034,A 180.000,B 0.000,C 180.000} C_DIS
LIN {X 123.005,Y 42.491,Z 55.032,A 180.000,B 0.000,C 180.000} C_DIS
LIN {X 122.879,Y 42.586,Z 55.029,A 180.000,B 0.000,C 180.000} C_DIS
LIN {X 122.749,Y 42.675,Z 55.027,A 180.000,B 0.000,C 180.000} C_DIS
LIN {X 122.487,Y 42.850,Z 55.022,A 180.000,B 0.000,C 180.000} C_DIS
LIN {X 122.216,Y 43.010,Z 55.018,A 180.000,B 0.000,C 180.000} C_DIS
LIN {X 121.939,Y 43.160,Z 55.014,A 180.000,B 0.000,C 180.000} C_DIS
LIN {X 121.657,Y 43.301,Z 55.011,A 180.000,B 0.000,C 180.000} C_DIS
LIN {X 121.368,Y 43.426,Z 55.008,A 180.000,B 0.000,C 180.000} C_DIS
LIN {X 121.074,Y 43.539,Z 55.005,A 180.000,B 0.000,C 180.000} C_DIS
LIN {X 120.777,Y 43.644,Z 55.003,A 180.000,B 0.000,C 180.000} C_DIS
LIN {X 120.474,Y 43.731,Z 55.002,A 180.000,B 0.000,C 180.000} C_DIS
LIN {X 120.169,Y 43.807,Z 55.001,A 180.000,B 0.000,C 180.000} C_DIS
LIN {X 119.861,Y 43.873,Z 55.000,A 180.000,B 0.000,C 180.000} C_DIS
LIN {X 119.632,Y 43.909,Z 55.000,A 180.000,B 0.000,C 180.000} C_DIS
; Cutting Move Starts
LIN {X 119.600,Y 43.914,Z 55.000,A 180.000,B 0.000,C 180.000} C_DIS
LIN {X 119.422,Y 43.941,Z 55.000,A 180.000,B 0.000,C 180.000} C_DIS
LIN {X 119.006,Y 43.981,Z 55.000,A 180.000,B 0.000,C 180.000} C_DIS
LIN {X 118.885,Y 43.987,Z 55.000,A 180.000,B 0.000,C 180.000} C_DIS
LIN {X 118.528,Y 43.998,Z 55.000,A 180.000,B 0.000,C 180.000} C_DIS
LIN {X 118.349,Y 43.994,Z 55.000,A 180.000,B 0.000,C 180.000} C_DIS
LIN {X 118.170,Y 43.988,Z 55.000,A 180.000,B 0.000,C 180.000} C_DIS
LIN {X 117.994,Y 43.981,Z 55.000,A 180.000,B 0.000,C 180.000} C_DIS
LIN {X 117.634,Y 43.947,Z 55.000,A 180.000,B 0.000,C 180.000} C_DIS
LIN {X 117.455,Y 43.923,Z 55.000,A 180.000,B 0.000,C 180.000} C_DIS
LIN {X 117.098,Y 43.866,Z 55.000,A 180.000,B 0.000,C 180.000} C_DIS
LIN {X 116.919,Y 43.827,Z 55.000,A 180.000,B 0.000,C 180.000} C_DIS
LIN {X 116.740,Y 43.787,Z 55.000,A 180.000,B 0.000,C 180.000} C_DIS
LIN {X 116.561,Y 43.742,Z 55.000,A 180.000,B 0.000,C 180.000} C_DIS
LIN {X 116.204,Y 43.638,Z 55.000,A 180.000,B 0.000,C 180.000} C_DIS
LIN {X 116.159,Y 43.623,Z 55.000,A 180.000,B 0.000,C 180.000} C_DIS
LIN {X 115.846,Y 43.511,Z 55.000,A 180.000,B 0.000,C 180.000} C_DIS
LIN {X 115.675,Y 43.444,Z 55.000,A 180.000,B 0.000,C 180.000} C_DIS
LIN {X 115.310,Y 43.286,Z 55.000,A 180.000,B 0.000,C 180.000} C_DIS
LIN {X 115.269,Y 43.266,Z 55.000,A 180.000,B 0.000,C 180.000} C_DIS
LIN {X 114.918,Y 43.087,Z 55.000,A 180.000,B 0.000,C 180.000} C_DIS
LIN {X 114.774,Y 43.004,Z 55.000,A 180.000,B 0.000,C 180.000} C_DIS
LIN {X 114.595,Y 42.898,Z 55.000,A 180.000,B 0.000,C 180.000} C_DIS
LIN {X 114.416,Y 42.787,Z 55.000,A 180.000,B 0.000,C 180.000} C_DIS
LIN {X 114.237,Y 42.665,Z 55.000,A 180.000,B 0.000,C 180.000} C_DIS
LIN {X 114.072,Y 42.550,Z 55.000,A 180.000,B 0.000,C 180.000} C_DIS
LIN {X 113.841,Y 42.372,Z 55.000,A 180.000,B 0.000,C 180.000} C_DIS
LIN {X 113.701,Y 42.261,Z 55.000,A 180.000,B 0.000,C 180.000} C_DIS
LIN {X 113.421,Y 42.014,Z 55.000,A 180.000,B 0.000,C 180.000} C_DIS
LIN {X 113.343,Y 41.943,Z 55.000,A 180.000,B 0.000,C 180.000} C_DIS
LIN {X 113.057,Y 41.657,Z 55.000,A 180.000,B 0.000,C 180.000} C_DIS
LIN {X 112.986,Y 41.579,Z 55.000,A 180.000,B 0.000,C 180.000} C_DIS
LIN {X 112.739,Y 41.299,Z 55.000,A 180.000,B 0.000,C 180.000} C_DIS
LIN {X 112.628,Y 41.159,Z 55.000,A 180.000,B 0.000,C 180.000} C_DIS
LIN {X 112.450,Y 40.928,Z 55.000,A 180.000,B 0.000,C 180.000} C_DIS
LIN {X 112.335,Y 40.763,Z 55.000,A 180.000,B 0.000,C 180.000} C_DIS
LIN {X 112.213,Y 40.584,Z 55.000,A 180.000,B 0.000,C 180.000} C_DIS
LIN {X 112.102,Y 40.405,Z 55.000,A 180.000,B 0.000,C 180.000} C_DIS
LIN {X 111.996,Y 40.226,Z 55.000,A 180.000,B 0.000,C 180.000} C_DIS
LIN {X 111.913,Y 40.082,Z 55.000,A 180.000,B 0.000,C 180.000} C_DIS
LIN {X 111.734,Y 39.731,Z 55.000,A 180.000,B 0.000,C 180.000} C_DIS
LIN {X 111.714,Y 39.690,Z 55.000,A 180.000,B 0.000,C 180.000} C_DIS
LIN {X 111.556,Y 39.325,Z 55.000,A 180.000,B 0.000,C 180.000} C_DIS
LIN {X 111.489,Y 39.154,Z 55.000,A 180.000,B 0.000,C 180.000} C_DIS
LIN {X 111.377,Y 38.841,Z 55.000,A 180.000,B 0.000,C 180.000} C_DIS
LIN {X 111.362,Y 38.796,Z 55.000,A 180.000,B 0.000,C 180.000} C_DIS
LIN {X 111.258,Y 38.439,Z 55.000,A 180.000,B 0.000,C 180.000} C_DIS
LIN {X 111.213,Y 38.260,Z 55.000,A 180.000,B 0.000,C 180.000} C_DIS
LIN {X 111.173,Y 38.081,Z 55.000,A 180.000,B 0.000,C 180.000} C_DIS
LIN {X 111.134,Y 37.902,Z 55.000,A 180.000,B 0.000,C 180.000} C_DIS
LIN {X 111.077,Y 37.545,Z 55.000,A 180.000,B 0.000,C 180.000} C_DIS
LIN {X 111.053,Y 37.366,Z 55.000,A 180.000,B 0.000,C 180.000} C_DIS
LIN {X 111.019,Y 37.006,Z 55.000,A 180.000,B 0.000,C 180.000} C_DIS
LIN {X 111.012,Y 36.830,Z 55.000,A 180.000,B 0.000,C 180.000} C_DIS
LIN {X 111.006,Y 36.651,Z 55.000,A 180.000,B 0.000,C 180.000} C_DIS
LIN {X 111.002,Y 36.472,Z 55.000,A 180.000,B 0.000,C 180.000} C_DIS
LIN {X 111.013,Y 36.115,Z 55.000,A 180.000,B 0.000,C 180.000} C_DIS
LIN {X 111.019,Y 35.994,Z 55.000,A 180.000,B 0.000,C 180.000} C_DIS
LIN {X 111.059,Y 35.578,Z 55.000,A 180.000,B 0.000,C 180.000} C_DIS
LIN {X 111.086,Y 35.400,Z 55.000,A 180.000,B 0.000,C 180.000} C_DIS
LIN {X 111.114,Y 35.221,Z 55.000,A 180.000,B 0.000,C 180.000} C_DIS
LIN {X 111.146,Y 35.042,Z 55.000,A 180.000,B 0.000,C 180.000} C_DIS
LIN {X 111.226,Y 34.685,Z 55.000,A 180.000,B 0.000,C 180.000} C_DIS
LIN {X 111.274,Y 34.506,Z 55.000,A 180.000,B 0.000,C 180.000} C_DIS
LIN {X 111.326,Y 34.327,Z 55.000,A 180.000,B 0.000,C 180.000} C_DIS
LIN {X 111.377,Y 34.159,Z 55.000,A 180.000,B 0.000,C 180.000} C_DIS
LIN {X 111.509,Y 33.791,Z 55.000,A 180.000,B 0.000,C 180.000} C_DIS
LIN {X 111.556,Y 33.675,Z 55.000,A 180.000,B 0.000,C 180.000} C_DIS
LIN {X 111.660,Y 33.433,Z 55.000,A 180.000,B 0.000,C 180.000} C_DIS
LIN {X 111.734,Y 33.269,Z 55.000,A 180.000,B 0.000,C 180.000} C_DIS
LIN {X 111.924,Y 32.897,Z 55.000,A 180.000,B 0.000,C 180.000} C_DIS
LIN {X 112.029,Y 32.718,Z 55.000,A 180.000,B 0.000,C 180.000} C_DIS
LIN {X 112.135,Y 32.539,Z 55.000,A 180.000,B 0.000,C 180.000} C_DIS
LIN {X 112.251,Y 32.361,Z 55.000,A 180.000,B 0.000,C 180.000} C_DIS
LIN {X 112.373,Y 32.182,Z 55.000,A 180.000,B 0.000,C 180.000} C_DIS
LIN {X 112.450,Y 32.072,Z 55.000,A 180.000,B 0.000,C 180.000} C_DIS
LIN {X 112.641,Y 31.824,Z 55.000,A 180.000,B 0.000,C 180.000} C_DIS
LIN {X 112.788,Y 31.646,Z 55.000,A 180.000,B 0.000,C 180.000} C_DIS
LIN {X 112.986,Y 31.421,Z 55.000,A 180.000,B 0.000,C 180.000} C_DIS
LIN {X 113.112,Y 31.288,Z 55.000,A 180.000,B 0.000,C 180.000} C_DIS
LIN {X 113.343,Y 31.057,Z 55.000,A 180.000,B 0.000,C 180.000} C_DIS
LIN {X 113.484,Y 30.930,Z 55.000,A 180.000,B 0.000,C 180.000} C_DIS
LIN {X 113.701,Y 30.739,Z 55.000,A 180.000,B 0.000,C 180.000} C_DIS
LIN {X 113.880,Y 30.598,Z 55.000,A 180.000,B 0.000,C 180.000} C_DIS
LIN {X 114.058,Y 30.460,Z 55.000,A 180.000,B 0.000,C 180.000} C_DIS
LIN {X 114.150,Y 30.394,Z 55.000,A 180.000,B 0.000,C 180.000} C_DIS
LIN {X 114.416,Y 30.213,Z 55.000,A 180.000,B 0.000,C 180.000} C_DIS
LIN {X 114.595,Y 30.102,Z 55.000,A 180.000,B 0.000,C 180.000} C_DIS
LIN {X 114.774,Y 29.996,Z 55.000,A 180.000,B 0.000,C 180.000} C_DIS
LIN {X 114.952,Y 29.896,Z 55.000,A 180.000,B 0.000,C 180.000} C_DIS
LIN {X 115.131,Y 29.805,Z 55.000,A 180.000,B 0.000,C 180.000} C_DIS
LIN {X 115.310,Y 29.714,Z 55.000,A 180.000,B 0.000,C 180.000} C_DIS
LIN {X 115.667,Y 29.559,Z 55.000,A 180.000,B 0.000,C 180.000} C_DIS
LIN {X 115.816,Y 29.500,Z 55.000,A 180.000,B 0.000,C 180.000} C_DIS
LIN {X 116.025,Y 29.425,Z 55.000,A 180.000,B 0.000,C 180.000} C_DIS
LIN {X 116.204,Y 29.362,Z 55.000,A 180.000,B 0.000,C 180.000} C_DIS
LIN {X 116.561,Y 29.258,Z 55.000,A 180.000,B 0.000,C 180.000} C_DIS
LIN {X 116.740,Y 29.213,Z 55.000,A 180.000,B 0.000,C 180.000} C_DIS
LIN {X 117.056,Y 29.143,Z 55.000,A 180.000,B 0.000,C 180.000} C_DIS
LIN {X 117.098,Y 29.134,Z 55.000,A 180.000,B 0.000,C 180.000} C_DIS
LIN {X 117.455,Y 29.077,Z 55.000,A 180.000,B 0.000,C 180.000} C_DIS
LIN {X 117.634,Y 29.053,Z 55.000,A 180.000,B 0.000,C 180.000} C_DIS
LIN {X 117.991,Y 29.020,Z 55.000,A 180.000,B 0.000,C 180.000} C_DIS
LIN {X 118.170,Y 29.012,Z 55.000,A 180.000,B 0.000,C 180.000} C_DIS
LIN {X 118.349,Y 29.006,Z 55.000,A 180.000,B 0.000,C 180.000} C_DIS
LIN {X 118.528,Y 29.002,Z 55.000,A 180.000,B 0.000,C 180.000} C_DIS
LIN {X 118.885,Y 29.013,Z 55.000,A 180.000,B 0.000,C 180.000} C_DIS
LIN {X 119.064,Y 29.025,Z 55.000,A 180.000,B 0.000,C 180.000} C_DIS
LIN {X 119.422,Y 29.059,Z 55.000,A 180.000,B 0.000,C 180.000} C_DIS
LIN {X 119.600,Y 29.086,Z 55.000,A 180.000,B 0.000,C 180.000} C_DIS
LIN {X 119.779,Y 29.114,Z 55.000,A 180.000,B 0.000,C 180.000} C_DIS
LIN {X 119.944,Y 29.143,Z 55.000,A 180.000,B 0.000,C 180.000} C_DIS
LIN {X 120.315,Y 29.226,Z 55.000,A 180.000,B 0.000,C 180.000} C_DIS
LIN {X 120.494,Y 29.274,Z 55.000,A 180.000,B 0.000,C 180.000} C_DIS
LIN {X 120.673,Y 29.326,Z 55.000,A 180.000,B 0.000,C 180.000} C_DIS
LIN {X 120.852,Y 29.381,Z 55.000,A 180.000,B 0.000,C 180.000} C_DIS
LIN {X 121.209,Y 29.509,Z 55.000,A 180.000,B 0.000,C 180.000} C_DIS
LIN {X 121.388,Y 29.583,Z 55.000,A 180.000,B 0.000,C 180.000} C_DIS
LIN {X 121.610,Y 29.679,Z 55.000,A 180.000,B 0.000,C 180.000} C_DIS
LIN {X 121.746,Y 29.742,Z 55.000,A 180.000,B 0.000,C 180.000} C_DIS
LIN {X 122.103,Y 29.924,Z 55.000,A 180.000,B 0.000,C 180.000} C_DIS
LIN {X 122.282,Y 30.029,Z 55.000,A 180.000,B 0.000,C 180.000} C_DIS
LIN {X 122.461,Y 30.135,Z 55.000,A 180.000,B 0.000,C 180.000} C_DIS
LIN {X 122.587,Y 30.215,Z 55.000,A 180.000,B 0.000,C 180.000} C_DIS
LIN {X 122.850,Y 30.394,Z 55.000,A 180.000,B 0.000,C 180.000} C_DIS
LIN {X 122.997,Y 30.503,Z 55.000,A 180.000,B 0.000,C 180.000} C_DIS
LIN {X 123.176,Y 30.641,Z 55.000,A 180.000,B 0.000,C 180.000} C_DIS
LIN {X 123.313,Y 30.752,Z 55.000,A 180.000,B 0.000,C 180.000} C_DIS
LIN {X 123.533,Y 30.945,Z 55.000,A 180.000,B 0.000,C 180.000} C_DIS
LIN {X 123.709,Y 31.109,Z 55.000,A 180.000,B 0.000,C 180.000} C_DIS
LIN {X 123.891,Y 31.291,Z 55.000,A 180.000,B 0.000,C 180.000} C_DIS
LIN {X 124.055,Y 31.467,Z 55.000,A 180.000,B 0.000,C 180.000} C_DIS
LIN {X 124.248,Y 31.687,Z 55.000,A 180.000,B 0.000,C 180.000} C_DIS
LIN {X 124.359,Y 31.824,Z 55.000,A 180.000,B 0.000,C 180.000} C_DIS
LIN {X 124.497,Y 32.003,Z 55.000,A 180.000,B 0.000,C 180.000} C_DIS
LIN {X 124.606,Y 32.150,Z 55.000,A 180.000,B 0.000,C 180.000} C_DIS
LIN {X 124.785,Y 32.413,Z 55.000,A 180.000,B 0.000,C 180.000} C_DIS
LIN {X 124.865,Y 32.539,Z 55.000,A 180.000,B 0.000,C 180.000} C_DIS
LIN {X 124.971,Y 32.718,Z 55.000,A 180.000,B 0.000,C 180.000} C_DIS
LIN {X 125.076,Y 32.897,Z 55.000,A 180.000,B 0.000,C 180.000} C_DIS
LIN {X 125.258,Y 33.254,Z 55.000,A 180.000,B 0.000,C 180.000} C_DIS
LIN {X 125.321,Y 33.390,Z 55.000,A 180.000,B 0.000,C 180.000} C_DIS
LIN {X 125.417,Y 33.612,Z 55.000,A 180.000,B 0.000,C 180.000} C_DIS
LIN {X 125.491,Y 33.791,Z 55.000,A 180.000,B 0.000,C 180.000} C_DIS
LIN {X 125.619,Y 34.148,Z 55.000,A 180.000,B 0.000,C 180.000} C_DIS
LIN {X 125.674,Y 34.327,Z 55.000,A 180.000,B 0.000,C 180.000} C_DIS
LIN {X 125.726,Y 34.506,Z 55.000,A 180.000,B 0.000,C 180.000} C_DIS
LIN {X 125.774,Y 34.685,Z 55.000,A 180.000,B 0.000,C 180.000} C_DIS
LIN {X 125.857,Y 35.056,Z 55.000,A 180.000,B 0.000,C 180.000} C_DIS
LIN {X 125.886,Y 35.221,Z 55.000,A 180.000,B 0.000,C 180.000} C_DIS
LIN {X 125.914,Y 35.400,Z 55.000,A 180.000,B 0.000,C 180.000} C_DIS
LIN {X 125.941,Y 35.578,Z 55.000,A 180.000,B 0.000,C 180.000} C_DIS
LIN {X 125.975,Y 35.936,Z 55.000,A 180.000,B 0.000,C 180.000} C_DIS
LIN {X 125.987,Y 36.115,Z 55.000,A 180.000,B 0.000,C 180.000} C_DIS
LIN {X 125.998,Y 36.472,Z 55.000,A 180.000,B 0.000,C 180.000} C_DIS
LIN {X 125.994,Y 36.651,Z 55.000,A 180.000,B 0.000,C 180.000} C_DIS
LIN {X 125.988,Y 36.830,Z 55.000,A 180.000,B 0.000,C 180.000} C_DIS
LIN {X 125.980,Y 37.009,Z 55.000,A 180.000,B 0.000,C 180.000} C_DIS
LIN {X 125.947,Y 37.366,Z 55.000,A 180.000,B 0.000,C 180.000} C_DIS
LIN {X 125.923,Y 37.545,Z 55.000,A 180.000,B 0.000,C 180.000} C_DIS
LIN {X 125.866,Y 37.902,Z 55.000,A 180.000,B 0.000,C 180.000} C_DIS
LIN {X 125.857,Y 37.944,Z 55.000,A 180.000,B 0.000,C 180.000} C_DIS
LIN {X 125.787,Y 38.260,Z 55.000,A 180.000,B 0.000,C 180.000} C_DIS
LIN {X 125.742,Y 38.439,Z 55.000,A 180.000,B 0.000,C 180.000} C_DIS
LIN {X 125.638,Y 38.796,Z 55.000,A 180.000,B 0.000,C 180.000} C_DIS
LIN {X 125.575,Y 38.975,Z 55.000,A 180.000,B 0.000,C 180.000} C_DIS
LIN {X 125.500,Y 39.184,Z 55.000,A 180.000,B 0.000,C 180.000} C_DIS
LIN {X 125.441,Y 39.333,Z 55.000,A 180.000,B 0.000,C 180.000} C_DIS
LIN {X 125.286,Y 39.690,Z 55.000,A 180.000,B 0.000,C 180.000} C_DIS
LIN {X 125.195,Y 39.869,Z 55.000,A 180.000,B 0.000,C 180.000} C_DIS
LIN {X 125.104,Y 40.048,Z 55.000,A 180.000,B 0.000,C 180.000} C_DIS
LIN {X 125.004,Y 40.226,Z 55.000,A 180.000,B 0.000,C 180.000} C_DIS
LIN {X 124.898,Y 40.405,Z 55.000,A 180.000,B 0.000,C 180.000} C_DIS
LIN {X 124.787,Y 40.584,Z 55.000,A 180.000,B 0.000,C 180.000} C_DIS
LIN {X 124.606,Y 40.850,Z 55.000,A 180.000,B 0.000,C 180.000} C_DIS
LIN {X 124.540,Y 40.942,Z 55.000,A 180.000,B 0.000,C 180.000} C_DIS
LIN {X 124.402,Y 41.120,Z 55.000,A 180.000,B 0.000,C 180.000} C_DIS
LIN {X 124.261,Y 41.299,Z 55.000,A 180.000,B 0.000,C 180.000} C_DIS
LIN {X 124.070,Y 41.516,Z 55.000,A 180.000,B 0.000,C 180.000} C_DIS
LIN {X 123.943,Y 41.657,Z 55.000,A 180.000,B 0.000,C 180.000} C_DIS
LIN {X 123.712,Y 41.888,Z 55.000,A 180.000,B 0.000,C 180.000} C_DIS
LIN {X 123.579,Y 42.014,Z 55.000,A 180.000,B 0.000,C 180.000} C_DIS
LIN {X 123.354,Y 42.212,Z 55.000,A 180.000,B 0.000,C 180.000} C_DIS
